LIN {X 0,Y 263.962,Z 436.135,A -85,B 0,C 180,E1 10063.892,E2 10063.892} C_VEL
LIN {X 0,Y 268.762,Z 444.869,A -85,B 0,C 180,E1 10060.552,E2 10060.552} C_VEL
LIN {X 0,Y 273.864,Z 454.801,A -85,B 0,C 180,E1 10057.516,E2 10057.516} C_VEL
LIN {X 0,Y 279.077,Z 465.837,A -85,B 0,C 180,E1 10054.772,E2 10054.772} C_VEL
LIN {X 0,Y 266.38,Z 615.165,A -85,B 0,C 180,E1 10051.274,E2 10051.274} C_VEL
LIN {X 0,Y 262.944,Z 636.67,A -85,B 0,C 180,E1 10050.519,E2 10050.519} C_VEL
LIN {X 0,Y 258.07,Z 657.385,A -85,B 0,C 180,E1 10049.523,E2 10049.523} C_VEL
LIN {X 0,Y 252.139,Z 676.761,A -85,B 0,C 180,E1 10048.274,E2 10048.274} C_VEL
LIN {X 0,Y 244.931,Z 696.333,A -85,B 0,C 180,E1 10046.572,E2 10046.572} C_VEL
LIN {X 0,Y 237.126,Z 714.604,A -85,B 0,C 180,E1 10044.466,E2 10044.466} C_VEL
LIN {X 0,Y 228.803,Z 731.913,A -85,B 0,C 180,E1 10041.866,E2 10041.866} C_VEL
LIN {X 0,Y 220.297,Z 748.012,A -85,B 0,C 180,E1 10038.744,E2 10038.744} C_VEL
LIN {X 0,Y 211.941,Z 762.843,A -85,B 0,C 180,E1 10035.042,E2 10035.042} C_VEL
LIN {X 0,Y 204.052,Z 776.444,A -85,B 0,C 180,E1 10030.668,E2 10030.668} C_VEL
LIN {X 0,Y 197.32,Z 788.149,A -85,B 0,C 180,E1 10025.831,E2 10025.831} C_VEL
LIN {X 0,Y 192.074,Z 797.92,A -85,B 0,C 180,E1 10020.673,E2 10020.673} C_VEL
LIN {X 0,Y 188.152,Z 806.55,A -85,B 0,C 180,E1 10014.822,E2 10014.822} C_VEL
LIN {X 0,Y 185.945,Z 813.61,A -85,B 0,C 180,E1 10008.496,E2 10008.496} C_VEL
LIN {X 0,Y 185.499,Z 818.499,A -85,B 0,C 180,E1 10002.451,E2 10002.451} C_VEL
LIN {X 0,Y 186.162,Z 821.531,A -85,B 0,C 180,E1 9996.786,E2 9996.786} C_VEL
LIN {X 0,Y 186.928,Z 822.719,A -85,B 0,C 180,E1 9992.146,E2 9992.146} C_VEL
LIN {X 0,Y 187.015,Z 822.81,A -85,B 0,C 180,E1 9988.759,E2 9988.759} C_VEL
LIN {X 0,Y 186.446,Z 822.014,A -85,B 0,C 180,E1 9984.769,E2 9984.769} C_VEL
LIN {X 0,Y 185.634,Z 819.662,A -85,B 0,C 180,E1 9979.448,E2 9979.448} C_VEL
LIN {X 0,Y 185.656,Z 815.362,A -85,B 0,C 180,E1 9973.416,E2 9973.416} C_VEL
LIN {X 0,Y 187.283,Z 808.876,A -85,B 0,C 180,E1 9967.063,E2 9967.063} C_VEL
LIN {X 0,Y 190.629,Z 800.812,A -85,B 0,C 180,E1 9961.149,E2 9961.149} C_VEL
LIN {X 0,Y 195.495,Z 791.337,A -85,B 0,C 180,E1 9955.766,E2 9955.766} C_VEL
LIN {X 0,Y 201.572,Z 780.562,A -85,B 0,C 180,E1 9950.954,E2 9950.954} C_VEL
LIN {X 0,Y 209.007,Z 767.743,A -85,B 0,C 180,E1 9946.46,E2 9946.46} C_VEL
LIN {X 0,Y 217.161,Z 753.439,A -85,B 0,C 180,E1 9942.553,E2 9942.553} C_VEL
LIN {X 0,Y 225.436,Z 738.145,A -85,B 0,C 180,E1 9939.292,E2 9939.292} C_VEL
LIN {X 0,Y 233.414,Z 722.238,A -85,B 0,C 180,E1 9936.636,E2 9936.636} C_VEL
LIN {X 0,Y 241.151,Z 705.141,A -85,B 0,C 180,E1 9934.404,E2 9934.404} C_VEL
LIN {X 0,Y 248.509,Z 686.643,A -85,B 0,C 180,E1 9932.554,E2 9932.554} C_VEL
LIN {X 0,Y 255.094,Z 667.118,A -85,B 0,C 180,E1 9931.085,E2 9931.085} C_VEL
LIN {X 0,Y 260.539,Z 647.028,A -85,B 0,C 180,E1 9929.966,E2 9929.966} C_VEL
LIN {X 0,Y 264.728,Z 625.774,A -85,B 0,C 180,E1 9929.09,E2 9929.09} C_VEL
LIN {X 0,Y 267.336,Z 604.079,A -85,B 0,C 180,E1 9928.456,E2 9928.456} C_VEL
LIN {X 0,Y 278.878,Z 465.633,A -85,B 0,C 180,E1 9925.226,E2 9925.226} C_VEL
LIN {X 0,Y 273.338,Z 453.94,A -85,B 0,C 180,E1 9922.303,E2 9922.303} C_VEL
LIN {X 0,Y 267.946,Z 443.512,A -85,B 0,C 180,E1 9919.057,E2 9919.057} C_VEL
LIN {X 0,Y 262.361,Z 433.364,A -85,B 0,C 180,E1 9915.019,E2 9915.019} C_VEL
LIN {X 0,Y 258.426,Z 426.882,A -85,B 0,C 180,E1 9911.493,E2 9911.493} C_VEL
LIN {X 0,Y 256.433,Z 423.717,A -85,B 0,C 180,E1 9909.312,E2 9909.312} C_VEL
LIN {X 0,Y 254.428,Z 420.112,A -85,B 0,C 180,E1 9906.543,E2 9906.543} C_VEL
LIN {X 0,Y 252.019,Z 415.913,A -85,B 0,C 180,E1 9901.364,E2 9901.364} C_VEL
LIN {X 0,Y 251.317,Z 414.93,A -85,B 0,C 180,E1 9895.664,E2 9895.664} C_VEL
LIN {X 0,Y 252.963,Z 416.019,A -85,B 0,C 180,E1 9889.754,E2 9889.754} C_VEL
LIN {X 0,Y 256.776,Z 421.342,A -85,B 0,C 180,E1 9883.95,E2 9883.95} C_VEL
LIN {X 0,Y 260.32,Z 426.562,A -85,B 0,C 180,E1 9880.361,E2 9880.361} C_VEL
LIN {X 0,Y 263.768,Z 431.814,A -85,B 0,C 180,E1 9877.547,E2 9877.547} C_VEL
LIN {X 0,Y 267.986,Z 438.368,A -85,B 0,C 180,E1 9874.65,E2 9874.65} C_VEL
LIN {X 0,Y 273.416,Z 447.764,A -85,B 0,C 180,E1 9871.435,E2 9871.435} C_VEL
LIN {X 0,Y 278.64,Z 457.79,A -85,B 0,C 180,E1 9868.724,E2 9868.724} C_VEL
LIN {X 0,Y 269.524,Z 577.471,A -85,B 0,C 180,E1 9866.054,E2 9866.054} C_VEL
LIN {X 0,Y 267.466,Z 596.812,A -85,B 0,C 180,E1 9865.36,E2 9865.36} C_VEL
LIN {X 0,Y 264.312,Z 615.233,A -85,B 0,C 180,E1 9864.419,E2 9864.419} C_VEL
LIN {X 0,Y 259.903,Z 633.791,A -85,B 0,C 180,E1 9863.145,E2 9863.145} C_VEL
LIN {X 0,Y 254.582,Z 651.308,A -85,B 0,C 180,E1 9861.583,E2 9861.583} C_VEL
LIN {X 0,Y 248.111,Z 668.635,A -85,B 0,C 180,E1 9859.608,E2 9859.608} C_VEL
LIN {X 0,Y 240.971,Z 684.785,A -85,B 0,C 180,E1 9857.257,E2 9857.257} C_VEL
LIN {X 0,Y 233.585,Z 699.288,A -85,B 0,C 180,E1 9854.586,E2 9854.586} C_VEL
LIN {X 0,Y 225.6,Z 713.172,A -85,B 0,C 180,E1 9851.327,E2 9851.327} C_VEL
LIN {X 0,Y 217.777,Z 725.421,A -85,B 0,C 180,E1 9847.634,E2 9847.634} C_VEL
LIN {X 0,Y 210.347,Z 736.116,A -85,B 0,C 180,E1 9843.461,E2 9843.461} C_VEL
LIN {X 0,Y 203.591,Z 745.264,A -85,B 0,C 180,E1 9838.769,E2 9838.769} C_VEL
LIN {X 0,Y 197.74,Z 752.844,A -85,B 0,C 180,E1 9833.544,E2 9833.544} C_VEL
LIN {X 0,Y 193.295,Z 758.557,A -85,B 0,C 180,E1 9828.081,E2 9828.081} C_VEL
LIN {X 0,Y 190.101,Z 762.723,A -85,B 0,C 180,E1 9822.145,E2 9822.145} C_VEL
LIN {X 0,Y 188.303,Z 765.165,A -85,B 0,C 180,E1 9816.096,E2 9816.096} C_VEL
LIN {X 0,Y 187.747,Z 765.976,A -85,B 0,C 180,E1 9810,E2 9810} C_VEL
LIN {X 0,Y 188.29,Z 765.2,A -85,B 0,C 180,E1 9803.904,E2 9803.904} C_VEL
LIN {X 0,Y 190.069,Z 762.799,A -85,B 0,C 180,E1 9797.853,E2 9797.853} C_VEL
LIN {X 0,Y 193.245,Z 758.673,A -85,B 0,C 180,E1 9791.915,E2 9791.915} C_VEL
LIN {X 0,Y 197.948,Z 752.674,A -85,B 0,C 180,E1 9786.167,E2 9786.167} C_VEL
LIN {X 0,Y 203.857,Z 745.036,A -85,B 0,C 180,E1 9780.951,E2 9780.951} C_VEL
LIN {X 0,Y 210.664,Z 735.828,A -85,B 0,C 180,E1 9776.269,E2 9776.269} C_VEL
LIN {X 0,Y 218.141,Z 725.064,A -85,B 0,C 180,E1 9772.108,E2 9772.108} C_VEL
LIN {X 0,Y 226.001,Z 712.736,A -85,B 0,C 180,E1 9768.425,E2 9768.425} C_VEL
LIN {X 0,Y 234.026,Z 698.729,A -85,B 0,C 180,E1 9765.172,E2 9765.172} C_VEL
LIN {X 0,Y 241.439,Z 684.148,A -85,B 0,C 180,E1 9762.513,E2 9762.513} C_VEL
LIN {X 0,Y 248.603,Z 667.849,A -85,B 0,C 180,E1 9760.17,E2 9760.17} C_VEL
LIN {X 0,Y 255.089,Z 650.314,A -85,B 0,C 180,E1 9758.199,E2 9758.199} C_VEL
LIN {X 0,Y 260.429,Z 632.572,A -85,B 0,C 180,E1 9756.641,E2 9756.641} C_VEL
LIN {X 0,Y 264.883,Z 613.37,A -85,B 0,C 180,E1 9755.356,E2 9755.356} C_VEL
LIN {X 0,Y 268.08,Z 593.774,A -85,B 0,C 180,E1 9754.394,E2 9754.394} C_VEL
LIN {X 0,Y 270.011,Z 573.44,A -85,B 0,C 180,E1 9753.717,E2 9753.717} C_VEL
LIN {X 0,Y 278.808,Z 457.69,A -85,B 0,C 180,E1 9751.152,E2 9751.152} C_VEL
LIN {X 0,Y 272.497,Z 445.95,A -85,B 0,C 180,E1 9747.839,E2 9747.839} C_VEL
LIN {X 0,Y 267.272,Z 437.11,A -85,B 0,C 180,E1 9744.653,E2 9744.653} C_VEL
LIN {X 0,Y 262.532,Z 429.641,A -85,B 0,C 180,E1 9741.212,E2 9741.212} C_VEL
LIN {X 0,Y 259.127,Z 424.746,A -85,B 0,C 180,E1 9738.213,E2 9738.213} C_VEL
LIN {X 0,Y 256.354,Z 420.667,A -85,B 0,C 180,E1 9735.149,E2 9735.149} C_VEL
LIN {X 0,Y 253.062,Z 416.095,A -85,B 0,C 180,E1 9729.782,E2 9729.782} C_VEL
LIN {X 0,Y 251.573,Z 415.164,A -85,B 0,C 180,E1 9723.875,E2 9723.875} C_VEL
LIN {X 0,Y 252.355,Z 416.185,A -85,B 0,C 180,E1 9718.411,E2 9718.411} C_VEL
LIN {X 0,Y 255.115,Z 421.076,A -85,B 0,C 180,E1 9712.796,E2 9712.796} C_VEL
LIN {X 0,Y 258.442,Z 426.742,A -85,B 0,C 180,E1 9708.734,E2 9708.734} C_VEL
LIN {X 0,Y 261.024,Z 431.187,A -85,B 0,C 180,E1 9706.272,E2 9706.272} C_VEL
LIN {X 0,Y 262.586,Z 435.115,A -85,B 0,C 180,E1 9704.85,E2 9704.85} C_VEL
LIN {X 0,Y 264.574,Z 443.488,A -85,B 0,C 180,E1 9702.933,E2 9702.933} C_VEL
LIN {X 0,Y 266.814,Z 452.064,A -85,B 0,C 180,E1 9701.05,E2 9701.05} C_VEL
LIN {X 0,Y 267.623,Z 454.063,A -85,B 0,C 180,E1 9700.49,E2 9700.49} C_VEL
LIN {X 0,Y 272.716,Z 464.616,A -85,B 0,C 180,E1 9697.416,E2 9697.416} C_VEL
LIN {X 0,Y 274.98,Z 470.078,A -85,B 0,C 180,E1 9696.14,E2 9696.14} C_VEL
LIN {X 0,Y 262.311,Z 614.422,A -85,B 0,C 180,E1 9692.779,E2 9692.779} C_VEL
LIN {X 0,Y 258.795,Z 635.834,A -85,B 0,C 180,E1 9692.035,E2 9692.035} C_VEL
LIN {X 0,Y 253.894,Z 656.209,A -85,B 0,C 180,E1 9691.07,E2 9691.07} C_VEL
LIN {X 0,Y 247.581,Z 676.274,A -85,B 0,C 180,E1 9689.793,E2 9689.793} C_VEL
LIN {X 0,Y 240.198,Z 695.651,A -85,B 0,C 180,E1 9688.12,E2 9688.12} C_VEL
LIN {X 0,Y 232.104,Z 713.934,A -85,B 0,C 180,E1 9686.019,E2 9686.019} C_VEL
LIN {X 0,Y 223.481,Z 731.176,A -85,B 0,C 180,E1 9683.423,E2 9683.423} C_VEL
LIN {X 0,Y 214.547,Z 747.362,A -85,B 0,C 180,E1 9680.258,E2 9680.258} C_VEL
LIN {X 0,Y 205.621,Z 762.427,A -85,B 0,C 180,E1 9676.428,E2 9676.428} C_VEL
LIN {X 0,Y 197.354,Z 775.9,A -85,B 0,C 180,E1 9671.969,E2 9671.969} C_VEL
LIN {X 0,Y 190.055,Z 787.822,A -85,B 0,C 180,E1 9666.85,E2 9666.85} C_VEL
LIN {X 0,Y 184.137,Z 798.176,A -85,B 0,C 180,E1 9661.053,E2 9661.053} C_VEL
LIN {X 0,Y 180.13,Z 806.495,A -85,B 0,C 180,E1 9654.951,E2 9654.951} C_VEL
LIN {X 0,Y 177.989,Z 812.955,A -85,B 0,C 180,E1 9648.674,E2 9648.674} C_VEL
LIN {X 0,Y 177.55,Z 817.657,A -85,B 0,C 180,E1 9642.356,E2 9642.356} C_VEL
LIN {X 0,Y 178.282,Z 820.523,A -85,B 0,C 180,E1 9636.44,E2 9636.44} C_VEL
LIN {X 0,Y 179.036,Z 821.548,A -85,B 0,C 180,E1 9631.92,E2 9631.92} C_VEL
LIN {X 0,Y 179.07,Z 821.577,A -85,B 0,C 180,E1 9628.4,E2 9628.4} C_VEL
LIN {X 0,Y 178.404,Z 820.702,A -85,B 0,C 180,E1 9624.21,E2 9624.21} C_VEL
LIN {X 0,Y 177.589,Z 818.027,A -85,B 0,C 180,E1 9618.306,E2 9618.306} C_VEL
LIN {X 0,Y 177.869,Z 813.516,A -85,B 0,C 180,E1 9611.991,E2 9611.991} C_VEL
LIN {X 0,Y 179.816,Z 807.245,A -85,B 0,C 180,E1 9605.703,E2 9605.703} C_VEL
LIN {X 0,Y 183.877,Z 798.609,A -85,B 0,C 180,E1 9599.261,E2 9599.261} C_VEL
LIN {X 0,Y 189.692,Z 788.341,A -85,B 0,C 180,E1 9593.445,E2 9593.445} C_VEL
LIN {X 0,Y 196.965,Z 776.407,A -85,B 0,C 180,E1 9588.263,E2 9588.263} C_VEL
LIN {X 0,Y 205.148,Z 763.047,A -85,B 0,C 180,E1 9583.795,E2 9583.795} C_VEL
LIN {X 0,Y 213.949,Z 748.192,A -85,B 0,C 180,E1 9579.968,E2 9579.968} C_VEL
LIN {X 0,Y 222.83,Z 732.143,A -85,B 0,C 180,E1 9576.782,E2 9576.782} C_VEL
LIN {X 0,Y 231.368,Z 715.151,A -85,B 0,C 180,E1 9574.18,E2 9574.18} C_VEL
LIN {X 0,Y 239.105,Z 697.83,A -85,B 0,C 180,E1 9572.138,E2 9572.138} C_VEL
LIN {X 0,Y 246.063,Z 679.96,A -85,B 0,C 180,E1 9570.524,E2 9570.524} C_VEL
LIN {X 0,Y 252.141,Z 661.532,A -85,B 0,C 180,E1 9569.264,E2 9569.264} C_VEL
LIN {X 0,Y 257.488,Z 640.986,A -85,B 0,C 180,E1 9568.212,E2 9568.212} C_VEL
LIN {X 0,Y 261.349,Z 619.931,A -85,B 0,C 180,E1 9567.418,E2 9567.418} C_VEL
LIN {X 0,Y 264.036,Z 594.652,A -85,B 0,C 180,E1 9566.746,E2 9566.746} C_VEL
LIN {X 0,Y 274.757,Z 469.441,A -85,B 0,C 180,E1 9563.824,E2 9563.824} C_VEL
LIN {X 0,Y 269.41,Z 457.799,A -85,B 0,C 180,E1 9560.758,E2 9560.758} C_VEL
LIN {X 0,Y 263.947,Z 447.113,A -85,B 0,C 180,E1 9557.129,E2 9557.129} C_VEL
LIN {X 0,Y 259.778,Z 439.543,A -85,B 0,C 180,E1 9553.805,E2 9553.805} C_VEL
LIN {X 0,Y 256.77,Z 434.226,A -85,B 0,C 180,E1 9550.886,E2 9550.886} C_VEL
LIN {X 0,Y 253.434,Z 428.163,A -85,B 0,C 180,E1 9546.569,E2 9546.569} C_VEL
LIN {X 0,Y 250.96,Z 423.8,A -85,B 0,C 180,E1 9541.141,E2 9541.141} C_VEL
LIN {X 0,Y 250.345,Z 422.871,A -85,B 0,C 180,E1 9535.647,E2 9535.647} C_VEL
LIN {X 0,Y 252.001,Z 423.991,A -85,B 0,C 180,E1 9529.714,E2 9529.714} C_VEL
LIN {X 0,Y 255.526,Z 429.237,A -85,B 0,C 180,E1 9524.219,E2 9524.219} C_VEL
LIN {X 0,Y 258.761,Z 434.142,A -85,B 0,C 180,E1 9520.825,E2 9520.825} C_VEL
LIN {X 0,Y 262.133,Z 439.449,A -85,B 0,C 180,E1 9517.971,E2 9517.971} C_VEL
LIN {X 0,Y 266.367,Z 446.383,A -85,B 0,C 180,E1 9514.961,E2 9514.961} C_VEL
LIN {X 0,Y 271.172,Z 455.032,A -85,B 0,C 180,E1 9512.017,E2 9512.017} C_VEL
LIN {X 0,Y 274.626,Z 461.918,A -85,B 0,C 180,E1 9510.11,E2 9510.11} C_VEL
LIN {X 0,Y 265.44,Z 578.24,A -85,B 0,C 180,E1 9507.518,E2 9507.518} C_VEL
LIN {X 0,Y 263.304,Z 597.581,A -85,B 0,C 180,E1 9506.825,E2 9506.825} C_VEL
LIN {X 0,Y 260.034,Z 616.06,A -85,B 0,C 180,E1 9505.886,E2 9505.886} C_VEL
LIN {X 0,Y 255.561,Z 634.361,A -85,B 0,C 180,E1 9504.639,E2 9504.639} C_VEL
LIN {X 0,Y 250.09,Z 651.862,A -85,B 0,C 180,E1 9503.09,E2 9503.09} C_VEL
LIN {X 0,Y 243.394,Z 669.282,A -85,B 0,C 180,E1 9501.118,E2 9501.118} C_VEL
LIN {X 0,Y 235.981,Z 685.526,A -85,B 0,C 180,E1 9498.762,E2 9498.762} C_VEL
LIN {X 0,Y 228.025,Z 700.565,A -85,B 0,C 180,E1 9495.98,E2 9495.98} C_VEL
LIN {X 0,Y 219.721,Z 714.42,A -85,B 0,C 180,E1 9492.689,E2 9492.689} C_VEL
LIN {X 0,Y 211.561,Z 726.652,A -85,B 0,C 180,E1 9488.944,E2 9488.944} C_VEL
LIN {X 0,Y 203.781,Z 737.336,A -85,B 0,C 180,E1 9484.69,E2 9484.69} C_VEL
LIN {X 0,Y 196.675,Z 746.477,A -85,B 0,C 180,E1 9479.881,E2 9479.881} C_VEL
LIN {X 0,Y 190.493,Z 754.053,A -85,B 0,C 180,E1 9474.497,E2 9474.497} C_VEL
LIN {X 0,Y 185.77,Z 759.763,A -85,B 0,C 180,E1 9468.84,E2 9468.84} C_VEL
LIN {X 0,Y 182.363,Z 763.927,A -85,B 0,C 180,E1 9462.668,E2 9462.668} C_VEL
LIN {X 0,Y 180.435,Z 766.367,A -85,B 0,C 180,E1 9456.363,E2 9456.363} C_VEL
LIN {X 0,Y 179.838,Z 767.178,A -85,B 0,C 180,E1 9450,E2 9450} C_VEL
LIN {X 0,Y 180.422,Z 766.402,A -85,B 0,C 180,E1 9443.637,E2 9443.637} C_VEL
LIN {X 0,Y 182.33,Z 764.002,A -85,B 0,C 180,E1 9437.329,E2 9437.329} C_VEL
LIN {X 0,Y 185.719,Z 759.877,A -85,B 0,C 180,E1 9431.155,E2 9431.155} C_VEL
LIN {X 0,Y 190.717,Z 753.881,A -85,B 0,C 180,E1 9425.203,E2 9425.203} C_VEL
LIN {X 0,Y 196.958,Z 746.25,A -85,B 0,C 180,E1 9419.831,E2 9419.831} C_VEL
LIN {X 0,Y 204.119,Z 737.048,A -85,B 0,C 180,E1 9415.034,E2 9415.034} C_VEL
LIN {X 0,Y 211.947,Z 726.296,A -85,B 0,C 180,E1 9410.793,E2 9410.793} C_VEL
LIN {X 0,Y 220.146,Z 713.986,A -85,B 0,C 180,E1 9407.059,E2 9407.059} C_VEL
LIN {X 0,Y 228.485,Z 700.025,A -85,B 0,C 180,E1 9403.778,E2 9403.778} C_VEL
LIN {X 0,Y 236.481,Z 684.837,A -85,B 0,C 180,E1 9401.002,E2 9401.002} C_VEL
LIN {X 0,Y 243.906,Z 668.454,A -85,B 0,C 180,E1 9398.657,E2 9398.657} C_VEL
LIN {X 0,Y 250.266,Z 651.876,A -85,B 0,C 180,E1 9396.793,E2 9396.793} C_VEL
LIN {X 0,Y 255.814,Z 634.148,A -85,B 0,C 180,E1 9395.228,E2 9395.228} C_VEL
LIN {X 0,Y 260.374,Z 615.388,A -85,B 0,C 180,E1 9393.96,E2 9393.96} C_VEL
LIN {X 0,Y 263.777,Z 595.743,A -85,B 0,C 180,E1 9392.979,E2 9392.979} C_VEL
LIN {X 0,Y 265.852,Z 575.618,A -85,B 0,C 180,E1 9392.291,E2 9392.291} C_VEL
LIN {X 0,Y 274.724,Z 461.747,A -85,B 0,C 180,E1 9389.729,E2 9389.729} C_VEL
LIN {X 0,Y 269.186,Z 451.135,A -85,B 0,C 180,E1 9386.589,E2 9386.589} C_VEL
LIN {X 0,Y 264.409,Z 442.959,A -85,B 0,C 180,E1 9383.454,E2 9383.454} C_VEL
LIN {X 0,Y 260.148,Z 436.17,A -85,B 0,C 180,E1 9380.12,E2 9380.12} C_VEL
LIN {X 0,Y 257.621,Z 432.313,A -85,B 0,C 180,E1 9377.739,E2 9377.739} C_VEL
LIN {X 0,Y 255.045,Z 428.396,A -85,B 0,C 180,E1 9374.763,E2 9374.763} C_VEL
LIN {X 0,Y 252.008,Z 423.989,A -85,B 0,C 180,E1 9369.593,E2 9369.593} C_VEL
LIN {X 0,Y 250.592,Z 423.106,A -85,B 0,C 180,E1 9363.661,E2 9363.661} C_VEL
LIN {X 0,Y 251.362,Z 424.279,A -85,B 0,C 180,E1 9358.405,E2 9358.405} C_VEL
LIN {X 0,Y 253.873,Z 428.918,A -85,B 0,C 180,E1 9353.101,E2 9353.101} C_VEL
LIN {X 0,Y 256.901,Z 434.265,A -85,B 0,C 180,E1 9349.233,E2 9349.233} C_VEL
LIN {X 0,Y 260.684,Z 440.814,A -85,B 0,C 180,E1 9345.621,E2 9345.621} C_VEL
LIN {X 0,Y 265.967,Z 450.804,A -85,B 0,C 180,E1 9341.592,E2 9341.592} C_VEL
LIN {X 0,Y 267.623,Z 454.063,A -85,B 0,C 180,E1 9340.49,E2 9340.49} C_VEL
LIN {X 0,Y 268.653,Z 457.702,A -85,B 0,C 180,E1 9339.728,E2 9339.728} C_VEL
LIN {X 0,Y 270.267,Z 470.787,A -85,B 0,C 180,E1 9338.119,E2 9338.119} C_VEL
LIN {X 0,Y 271.051,Z 473.538,A -85,B 0,C 180,E1 9337.597,E2 9337.597} C_VEL
LIN {X 0,Y 258.457,Z 613.492,A -85,B 0,C 180,E1 9334.336,E2 9334.336} C_VEL
LIN {X 0,Y 254.871,Z 634.831,A -85,B 0,C 180,E1 9333.607,E2 9333.607} C_VEL
LIN {X 0,Y 249.872,Z 655.168,A -85,B 0,C 180,E1 9332.661,E2 9332.661} C_VEL
LIN {X 0,Y 243.592,Z 674.701,A -85,B 0,C 180,E1 9331.446,E2 9331.446} C_VEL
LIN {X 0,Y 235.986,Z 694.185,A -85,B 0,C 180,E1 9329.804,E2 9329.804} C_VEL
LIN {X 0,Y 227.614,Z 712.526,A -85,B 0,C 180,E1 9327.735,E2 9327.735} C_VEL
LIN {X 0,Y 218.527,Z 730.074,A -85,B 0,C 180,E1 9325.116,E2 9325.116} C_VEL
LIN {X 0,Y 209.154,Z 746.368,A -85,B 0,C 180,E1 9321.926,E2 9321.926} C_VEL
LIN {X 0,Y 199.978,Z 761.113,A -85,B 0,C 180,E1 9318.155,E2 9318.155} C_VEL
LIN {X 0,Y 191.242,Z 774.603,A -85,B 0,C 180,E1 9313.639,E2 9313.639} C_VEL
LIN {X 0,Y 183.44,Z 786.534,A -85,B 0,C 180,E1 9308.415,E2 9308.415} C_VEL
LIN {X 0,Y 177.041,Z 796.897,A -85,B 0,C 180,E1 9302.446,E2 9302.446} C_VEL
LIN {X 0,Y 172.62,Z 805.225,A -85,B 0,C 180,E1 9296.116,E2 9296.116} C_VEL
LIN {X 0,Y 170.181,Z 811.698,A -85,B 0,C 180,E1 9289.565,E2 9289.565} C_VEL
LIN {X 0,Y 169.577,Z 816.415,A -85,B 0,C 180,E1 9282.947,E2 9282.947} C_VEL
LIN {X 0,Y 170.287,Z 819.301,A -85,B 0,C 180,E1 9276.744,E2 9276.744} C_VEL
LIN {X 0,Y 171.107,Z 820.343,A -85,B 0,C 180,E1 9272.009,E2 9272.009} C_VEL
LIN {X 0,Y 171.178,Z 820.405,A -85,B 0,C 180,E1 9268.661,E2 9268.661} C_VEL
LIN {X 0,Y 170.476,Z 819.577,A -85,B 0,C 180,E1 9264.278,E2 9264.278} C_VEL
LIN {X 0,Y 169.621,Z 816.985,A -85,B 0,C 180,E1 9258.094,E2 9258.094} C_VEL
LIN {X 0,Y 169.97,Z 812.559,A -85,B 0,C 180,E1 9251.479,E2 9251.479} C_VEL
LIN {X 0,Y 172.273,Z 805.975,A -85,B 0,C 180,E1 9244.566,E2 9244.566} C_VEL
LIN {X 0,Y 176.757,Z 797.329,A -85,B 0,C 180,E1 9237.879,E2 9237.879} C_VEL
LIN {X 0,Y 183.113,Z 786.955,A -85,B 0,C 180,E1 9231.839,E2 9231.839} C_VEL
LIN {X 0,Y 190.759,Z 775.213,A -85,B 0,C 180,E1 9226.637,E2 9226.637} C_VEL
LIN {X 0,Y 199.421,Z 761.827,A -85,B 0,C 180,E1 9222.096,E2 9222.096} C_VEL
LIN {X 0,Y 208.727,Z 746.868,A -85,B 0,C 180,E1 9218.225,E2 9218.225} C_VEL
LIN {X 0,Y 217.99,Z 730.79,A -85,B 0,C 180,E1 9215.045,E2 9215.045} C_VEL
LIN {X 0,Y 226.895,Z 713.67,A -85,B 0,C 180,E1 9212.45,E2 9212.45} C_VEL
LIN {X 0,Y 235.227,Z 695.538,A -85,B 0,C 180,E1 9210.362,E2 9210.362} C_VEL
LIN {X 0,Y 242.416,Z 677.385,A -85,B 0,C 180,E1 9208.784,E2 9208.784} C_VEL
LIN {X 0,Y 248.711,Z 658.403,A -85,B 0,C 180,E1 9207.548,E2 9207.548} C_VEL
LIN {X 0,Y 253.921,Z 638.253,A -85,B 0,C 180,E1 9206.563,E2 9206.563} C_VEL
LIN {X 0,Y 257.673,Z 617.588,A -85,B 0,C 180,E1 9205.814,E2 9205.814} C_VEL
LIN {X 0,Y 260.622,Z 589.211,A -85,B 0,C 180,E1 9205.086,E2 9205.086} C_VEL
LIN {X 0,Y 270.847,Z 473.338,A -85,B 0,C 180,E1 9202.405,E2 9202.405} C_VEL
LIN {X 0,Y 266.038,Z 462.77,A -85,B 0,C 180,E1 9199.427,E2 9199.427} C_VEL
LIN {X 0,Y 261.467,Z 453.484,A -85,B 0,C 180,E1 9196.152,E2 9196.152} C_VEL
LIN {X 0,Y 257.896,Z 446.68,A -85,B 0,C 180,E1 9193.109,E2 9193.109} C_VEL
LIN {X 0,Y 254.958,Z 441.205,A -85,B 0,C 180,E1 9190.05,E2 9190.05} C_VEL
LIN {X 0,Y 251.865,Z 435.512,A -85,B 0,C 180,E1 9185.695,E2 9185.695} C_VEL
LIN {X 0,Y 249.905,Z 431.687,A -85,B 0,C 180,E1 9180.917,E2 9180.917} C_VEL
LIN {X 0,Y 249.389,Z 430.818,A -85,B 0,C 180,E1 9175.4,E2 9175.4} C_VEL
LIN {X 0,Y 250.937,Z 431.891,A -85,B 0,C 180,E1 9169.902,E2 9169.902} C_VEL
LIN {X 0,Y 254.192,Z 436.961,A -85,B 0,C 180,E1 9164.602,E2 9164.602} C_VEL
LIN {X 0,Y 257.218,Z 441.719,A -85,B 0,C 180,E1 9161.295,E2 9161.295} C_VEL
LIN {X 0,Y 260.737,Z 447.429,A -85,B 0,C 180,E1 9158.221,E2 9158.221} C_VEL
LIN {X 0,Y 265.223,Z 455.175,A -85,B 0,C 180,E1 9154.965,E2 9154.965} C_VEL
LIN {X 0,Y 270.149,Z 464.689,A -85,B 0,C 180,E1 9151.902,E2 9151.902} C_VEL
LIN {X 0,Y 270.764,Z 466.184,A -85,B 0,C 180,E1 9151.534,E2 9151.534} C_VEL
LIN {X 0,Y 261.543,Z 578.893,A -85,B 0,C 180,E1 9149.031,E2 9149.031} C_VEL
LIN {X 0,Y 259.335,Z 598.253,A -85,B 0,C 180,E1 9148.341,E2 9148.341} C_VEL
LIN {X 0,Y 256.033,Z 616.456,A -85,B 0,C 180,E1 9147.426,E2 9147.426} C_VEL
LIN {X 0,Y 251.465,Z 634.7,A -85,B 0,C 180,E1 9146.2,E2 9146.2} C_VEL
LIN {X 0,Y 245.442,Z 653.314,A -85,B 0,C 180,E1 9144.559,E2 9144.559} C_VEL
LIN {X 0,Y 238.524,Z 670.647,A -85,B 0,C 180,E1 9142.592,E2 9142.592} C_VEL
LIN {X 0,Y 230.865,Z 686.815,A -85,B 0,C 180,E1 9140.239,E2 9140.239} C_VEL
LIN {X 0,Y 222.606,Z 701.837,A -85,B 0,C 180,E1 9137.443,E2 9137.443} C_VEL
LIN {X 0,Y 213.973,Z 715.667,A -85,B 0,C 180,E1 9134.125,E2 9134.125} C_VEL
LIN {X 0,Y 205.461,Z 727.883,A -85,B 0,C 180,E1 9130.332,E2 9130.332} C_VEL
LIN {X 0,Y 197.315,Z 738.556,A -85,B 0,C 180,E1 9126.001,E2 9126.001} C_VEL
LIN {X 0,Y 189.838,Z 747.69,A -85,B 0,C 180,E1 9121.074,E2 9121.074} C_VEL
LIN {X 0,Y 183.302,Z 755.261,A -85,B 0,C 180,E1 9115.525,E2 9115.525} C_VEL
LIN {X 0,Y 178.101,Z 761.156,A -85,B 0,C 180,E1 9109.41,E2 9109.41} C_VEL
LIN {X 0,Y 174.64,Z 765.131,A -85,B 0,C 180,E1 9103.239,E2 9103.239} C_VEL
LIN {X 0,Y 172.572,Z 767.569,A -85,B 0,C 180,E1 9096.654,E2 9096.654} C_VEL
LIN {X 0,Y 171.929,Z 768.379,A -85,B 0,C 180,E1 9090,E2 9090} C_VEL
LIN {X 0,Y 172.558,Z 767.603,A -85,B 0,C 180,E1 9083.345,E2 9083.345} C_VEL
LIN {X 0,Y 174.606,Z 765.204,A -85,B 0,C 180,E1 9076.759,E2 9076.759} C_VEL
LIN {X 0,Y 178.23,Z 761.081,A -85,B 0,C 180,E1 9070.331,E2 9070.331} C_VEL
LIN {X 0,Y 183.543,Z 755.089,A -85,B 0,C 180,E1 9064.165,E2 9064.165} C_VEL
LIN {X 0,Y 190.141,Z 747.462,A -85,B 0,C 180,E1 9058.629,E2 9058.629} C_VEL
LIN {X 0,Y 197.674,Z 738.268,A -85,B 0,C 180,E1 9053.716,E2 9053.716} C_VEL
LIN {X 0,Y 205.871,Z 727.526,A -85,B 0,C 180,E1 9049.4,E2 9049.4} C_VEL
LIN {X 0,Y 214.422,Z 715.233,A -85,B 0,C 180,E1 9045.618,E2 9045.618} C_VEL
LIN {X 0,Y 223.091,Z 701.302,A -85,B 0,C 180,E1 9042.313,E2 9042.313} C_VEL
LIN {X 0,Y 231.381,Z 686.158,A -85,B 0,C 180,E1 9039.527,E2 9039.527} C_VEL
LIN {X 0,Y 239.064,Z 669.839,A -85,B 0,C 180,E1 9037.182,E2 9037.182} C_VEL
LIN {X 0,Y 245.998,Z 652.299,A -85,B 0,C 180,E1 9035.22,E2 9035.22} C_VEL
LIN {X 0,Y 251.698,Z 634.574,A -85,B 0,C 180,E1 9033.674,E2 9033.674} C_VEL
LIN {X 0,Y 256.472,Z 615.362,A -85,B 0,C 180,E1 9032.396,E2 9032.396} C_VEL
LIN {X 0,Y 259.942,Z 595.562,A -85,B 0,C 180,E1 9031.429,E2 9031.429} C_VEL
LIN {X 0,Y 262.042,Z 575.244,A -85,B 0,C 180,E1 9030.751,E2 9030.751} C_VEL
LIN {X 0,Y 270.904,Z 465.97,A -85,B 0,C 180,E1 9028.313,E2 9028.313} C_VEL
LIN {X 0,Y 265.845,Z 456.132,A -85,B 0,C 180,E1 9025.211,E2 9025.211} C_VEL
LIN {X 0,Y 261.321,Z 448.177,A -85,B 0,C 180,E1 9021.964,E2 9021.964} C_VEL
LIN {X 0,Y 257.639,Z 442.271,A -85,B 0,C 180,E1 9018.791,E2 9018.791} C_VEL
LIN {X 0,Y 255.622,Z 439.169,A -85,B 0,C 180,E1 9016.708,E2 9016.708} C_VEL
LIN {X 0,Y 253.747,Z 436.123,A -85,B 0,C 180,E1 9014.374,E2 9014.374} C_VEL
LIN {X 0,Y 250.952,Z 431.883,A -85,B 0,C 180,E1 9009.402,E2 9009.402} C_VEL
LIN {X 0,Y 249.613,Z 431.063,A -85,B 0,C 180,E1 9003.445,E2 9003.445} C_VEL
LIN {X 0,Y 250.31,Z 432.173,A -85,B 0,C 180,E1 8998.627,E2 8998.627} C_VEL
LIN {X 0,Y 252.595,Z 436.657,A -85,B 0,C 180,E1 8993.482,E2 8993.482} C_VEL
LIN {X 0,Y 255.473,Z 441.965,A -85,B 0,C 180,E1 8989.629,E2 8989.629} C_VEL
LIN {X 0,Y 259.181,Z 448.801,A -85,B 0,C 180,E1 8985.934,E2 8985.934} C_VEL
LIN {X 0,Y 263.838,Z 457.95,A -85,B 0,C 180,E1 8982.238,E2 8982.238} C_VEL
LIN {X 0,Y 268.608,Z 468.029,A -85,B 0,C 180,E1 8979.063,E2 8979.063} C_VEL
LIN {X 0,Y 271.051,Z 473.538,A -85,B 0,C 180,E1 8977.597,E2 8977.597} C_VEL
LIN {X 0,Y 271.539,Z 476.413,A -85,B 0,C 180,E1 8977.208,E2 8977.208} C_VEL
LIN {X 0,Y 271.269,Z 480.92,A -85,B 0,C 180,E1 8977.051,E2 8977.051} C_VEL
LIN {X 0,Y 269.93,Z 487.325,A -85,B 0,C 180,E1 8977.239,E2 8977.239} C_VEL
LIN {X 0,Y 265.57,Z 502.194,A -85,B 0,C 180,E1 8978.257,E2 8978.257} C_VEL
LIN {X 0,Y 264.534,Z 508.324,A -85,B 0,C 180,E1 8978.34,E2 8978.34} C_VEL
LIN {X 0,Y 254.757,Z 612.84,A -85,B 0,C 180,E1 8975.931,E2 8975.931} C_VEL
LIN {X 0,Y 251.088,Z 634.078,A -85,B 0,C 180,E1 8975.216,E2 8975.216} C_VEL
LIN {X 0,Y 245.844,Z 654.788,A -85,B 0,C 180,E1 8974.266,E2 8974.266} C_VEL
LIN {X 0,Y 239.415,Z 674.224,A -85,B 0,C 180,E1 8973.075,E2 8973.075} C_VEL
LIN {X 0,Y 231.603,Z 693.598,A -85,B 0,C 180,E1 8971.463,E2 8971.463} C_VEL
LIN {X 0,Y 222.975,Z 711.859,A -85,B 0,C 180,E1 8969.422,E2 8969.422} C_VEL
LIN {X 0,Y 213.717,Z 729.073,A -85,B 0,C 180,E1 8966.868,E2 8966.868} C_VEL
LIN {X 0,Y 204.038,Z 745.225,A -85,B 0,C 180,E1 8963.715,E2 8963.715} C_VEL
LIN {X 0,Y 194.533,Z 759.801,A -85,B 0,C 180,E1 8959.979,E2 8959.979} C_VEL
LIN {X 0,Y 185.3,Z 773.305,A -85,B 0,C 180,E1 8955.417,E2 8955.417} C_VEL
LIN {X 0,Y 176.976,Z 785.247,A -85,B 0,C 180,E1 8950.094,E2 8950.094} C_VEL
LIN {X 0,Y 170.06,Z 795.62,A -85,B 0,C 180,E1 8943.954,E2 8943.954} C_VEL
LIN {X 0,Y 165.185,Z 803.954,A -85,B 0,C 180,E1 8937.388,E2 8937.388} C_VEL
LIN {X 0,Y 162.407,Z 810.439,A -85,B 0,C 180,E1 8930.543,E2 8930.543} C_VEL
LIN {X 0,Y 161.613,Z 815.173,A -85,B 0,C 180,E1 8923.597,E2 8923.597} C_VEL
LIN {X 0,Y 162.282,Z 818.076,A -85,B 0,C 180,E1 8917.078,E2 8917.078} C_VEL
LIN {X 0,Y 163.175,Z 819.137,A -85,B 0,C 180,E1 8912.107,E2 8912.107} C_VEL
LIN {X 0,Y 163.256,Z 819.202,A -85,B 0,C 180,E1 8908.596,E2 8908.596} C_VEL
LIN {X 0,Y 162.481,Z 818.356,A -85,B 0,C 180,E1 8903.995,E2 8903.995} C_VEL
LIN {X 0,Y 161.638,Z 815.742,A -85,B 0,C 180,E1 8897.497,E2 8897.497} C_VEL
LIN {X 0,Y 162.159,Z 811.3,A -85,B 0,C 180,E1 8890.552,E2 8890.552} C_VEL
LIN {X 0,Y 164.796,Z 804.703,A -85,B 0,C 180,E1 8883.323,E2 8883.323} C_VEL
LIN {X 0,Y 169.748,Z 796.048,A -85,B 0,C 180,E1 8876.381,E2 8876.381} C_VEL
LIN {X 0,Y 176.556,Z 785.763,A -85,B 0,C 180,E1 8870.215,E2 8870.215} C_VEL
LIN {X 0,Y 184.79,Z 773.917,A -85,B 0,C 180,E1 8864.863,E2 8864.863} C_VEL
LIN {X 0,Y 193.946,Z 760.519,A -85,B 0,C 180,E1 8860.273,E2 8860.273} C_VEL
LIN {X 0,Y 203.708,Z 745.539,A -85,B 0,C 180,E1 8856.396,E2 8856.396} C_VEL
LIN {X 0,Y 213.209,Z 729.692,A -85,B 0,C 180,E1 8853.276,E2 8853.276} C_VEL
LIN {X 0,Y 222.597,Z 712.279,A -85,B 0,C 180,E1 8850.666,E2 8850.666} C_VEL
LIN {X 0,Y 231.206,Z 694.085,A -85,B 0,C 180,E1 8848.615,E2 8848.615} C_VEL
LIN {X 0,Y 238.607,Z 675.837,A -85,B 0,C 180,E1 8847.072,E2 8847.072} C_VEL
LIN {X 0,Y 245.023,Z 656.831,A -85,B 0,C 180,E1 8845.873,E2 8845.873} C_VEL
LIN {X 0,Y 250.242,Z 636.931,A -85,B 0,C 180,E1 8844.927,E2 8844.927} C_VEL
LIN {X 0,Y 254.035,Z 616.367,A -85,B 0,C 180,E1 8844.2,E2 8844.2} C_VEL
LIN {X 0,Y 257.092,Z 587.514,A -85,B 0,C 180,E1 8843.472,E2 8843.472} C_VEL
LIN {X 0,Y 267.095,Z 477.349,A -85,B 0,C 180,E1 8840.946,E2 8840.946} C_VEL
LIN {X 0,Y 262.464,Z 466.849,A -85,B 0,C 180,E1 8837.801,E2 8837.801} C_VEL
LIN {X 0,Y 257.967,Z 457.509,A -85,B 0,C 180,E1 8834.19,E2 8834.19} C_VEL
LIN {X 0,Y 254.309,Z 450.317,A -85,B 0,C 180,E1 8830.534,E2 8830.534} C_VEL
LIN {X 0,Y 252.182,Z 446.451,A -85,B 0,C 180,E1 8827.861,E2 8827.861} C_VEL
LIN {X 0,Y 250.603,Z 443.213,A -85,B 0,C 180,E1 8825.265,E2 8825.265} C_VEL
LIN {X 0,Y 248.856,Z 439.575,A -85,B 0,C 180,E1 8820.69,E2 8820.69} C_VEL
LIN {X 0,Y 248.41,Z 438.758,A -85,B 0,C 180,E1 8815.382,E2 8815.382} C_VEL
LIN {X 0,Y 249.865,Z 439.829,A -85,B 0,C 180,E1 8810.091,E2 8810.091} C_VEL
LIN {X 0,Y 252.865,Z 444.683,A -85,B 0,C 180,E1 8804.989,E2 8804.989} C_VEL
LIN {X 0,Y 255.69,Z 449.295,A -85,B 0,C 180,E1 8801.769,E2 8801.769} C_VEL
LIN {X 0,Y 259.434,Z 455.525,A -85,B 0,C 180,E1 8798.404,E2 8798.404} C_VEL
LIN {X 0,Y 264.142,Z 464.247,A -85,B 0,C 180,E1 8794.915,E2 8794.915} C_VEL
LIN {X 0,Y 267.074,Z 470.47,A -85,B 0,C 180,E1 8792.997,E2 8792.997} C_VEL
LIN {X 0,Y 257.843,Z 579.44,A -85,B 0,C 180,E1 8790.592,E2 8790.592} C_VEL
LIN {X 0,Y 255.589,Z 598.711,A -85,B 0,C 180,E1 8789.912,E2 8789.912} C_VEL
LIN {X 0,Y 252.035,Z 617.628,A -85,B 0,C 180,E1 8788.968,E2 8788.968} C_VEL
LIN {X 0,Y 247.178,Z 636.274,A -85,B 0,C 180,E1 8787.715,E2 8787.715} C_VEL
LIN {X 0,Y 241.308,Z 653.871,A -85,B 0,C 180,E1 8786.175,E2 8786.175} C_VEL
LIN {X 0,Y 234.158,Z 671.292,A -85,B 0,C 180,E1 8784.221,E2 8784.221} C_VEL
LIN {X 0,Y 226.228,Z 687.532,A -85,B 0,C 180,E1 8781.877,E2 8781.877} C_VEL
LIN {X 0,Y 217.745,Z 702.468,A -85,B 0,C 180,E1 8779.116,E2 8779.116} C_VEL
LIN {X 0,Y 208.949,Z 716.095,A -85,B 0,C 180,E1 8775.869,E2 8775.869} C_VEL
LIN {X 0,Y 200.025,Z 728.437,A -85,B 0,C 180,E1 8772.052,E2 8772.052} C_VEL
LIN {X 0,Y 191.434,Z 739.221,A -85,B 0,C 180,E1 8767.667,E2 8767.667} C_VEL
LIN {X 0,Y 183.495,Z 748.46,A -85,B 0,C 180,E1 8762.645,E2 8762.645} C_VEL
LIN {X 0,Y 176.504,Z 756.135,A -85,B 0,C 180,E1 8756.947,E2 8756.947} C_VEL
LIN {X 0,Y 170.775,Z 762.231,A -85,B 0,C 180,E1 8750.481,E2 8750.481} C_VEL
LIN {X 0,Y 166.936,Z 766.334,A -85,B 0,C 180,E1 8743.861,E2 8743.861} C_VEL
LIN {X 0,Y 164.713,Z 768.772,A -85,B 0,C 180,E1 8736.973,E2 8736.973} C_VEL
LIN {X 0,Y 164.019,Z 769.581,A -85,B 0,C 180,E1 8730,E2 8730} C_VEL
LIN {X 0,Y 164.698,Z 768.805,A -85,B 0,C 180,E1 8723.026,E2 8723.026} C_VEL
LIN {X 0,Y 167.009,Z 766.307,A -85,B 0,C 180,E1 8715.902,E2 8715.902} C_VEL
LIN {X 0,Y 171.022,Z 762.045,A -85,B 0,C 180,E1 8709.107,E2 8709.107} C_VEL
LIN {X 0,Y 176.764,Z 755.939,A -85,B 0,C 180,E1 8702.732,E2 8702.732} C_VEL
LIN {X 0,Y 183.818,Z 748.206,A -85,B 0,C 180,E1 8697.049,E2 8697.049} C_VEL
LIN {X 0,Y 191.816,Z 738.903,A -85,B 0,C 180,E1 8692.043,E2 8692.043} C_VEL
LIN {X 0,Y 200.458,Z 728.045,A -85,B 0,C 180,E1 8687.674,E2 8687.674} C_VEL
LIN {X 0,Y 209.421,Z 715.62,A -85,B 0,C 180,E1 8683.87,E2 8683.87} C_VEL
LIN {X 0,Y 218.16,Z 702.06,A -85,B 0,C 180,E1 8680.669,E2 8680.669} C_VEL
LIN {X 0,Y 226.765,Z 686.843,A -85,B 0,C 180,E1 8677.887,E2 8677.887} C_VEL
LIN {X 0,Y 234.719,Z 670.442,A -85,B 0,C 180,E1 8675.551,E2 8675.551} C_VEL
LIN {X 0,Y 241.595,Z 653.631,A -85,B 0,C 180,E1 8673.682,E2 8673.682} C_VEL
LIN {X 0,Y 247.56,Z 635.707,A -85,B 0,C 180,E1 8672.124,E2 8672.124} C_VEL
LIN {X 0,Y 252.462,Z 616.691,A -85,B 0,C 180,E1 8670.863,E2 8670.863} C_VEL
LIN {X 0,Y 256.095,Z 596.836,A -85,B 0,C 180,E1 8669.893,E2 8669.893} C_VEL
LIN {X 0,Y 258.309,Z 576.478,A -85,B 0,C 180,E1 8669.21,E2 8669.21} C_VEL
LIN {X 0,Y 267.24,Z 470.279,A -85,B 0,C 180,E1 8666.858,E2 8666.858} C_VEL
LIN {X 0,Y 262.656,Z 461.236,A -85,B 0,C 180,E1 8663.799,E2 8663.799} C_VEL
LIN {X 0,Y 258.568,Z 454.007,A -85,B 0,C 180,E1 8660.603,E2 8660.603} C_VEL
LIN {X 0,Y 255.072,Z 447.992,A -85,B 0,C 180,E1 8657.215,E2 8657.215} C_VEL
LIN {X 0,Y 252.461,Z 443.849,A -85,B 0,C 180,E1 8653.981,E2 8653.981} C_VEL
LIN {X 0,Y 249.889,Z 439.776,A -85,B 0,C 180,E1 8649.21,E2 8649.21} C_VEL
LIN {X 0,Y 248.64,Z 439.004,A -85,B 0,C 180,E1 8643.459,E2 8643.459} C_VEL
LIN {X 0,Y 249.26,Z 440.065,A -85,B 0,C 180,E1 8638.851,E2 8638.851} C_VEL
LIN {X 0,Y 251.292,Z 444.281,A -85,B 0,C 180,E1 8633.948,E2 8633.948} C_VEL
LIN {X 0,Y 254.152,Z 449.837,A -85,B 0,C 180,E1 8629.918,E2 8629.918} C_VEL
LIN {X 0,Y 257.809,Z 457,A -85,B 0,C 180,E1 8626.144,E2 8626.144} C_VEL
LIN {X 0,Y 261.951,Z 465.547,A -85,B 0,C 180,E1 8622.737,E2 8622.737} C_VEL
LIN {X 0,Y 266.413,Z 475.424,A -85,B 0,C 180,E1 8619.63,E2 8619.63} C_VEL
LIN {X 0,Y 267.328,Z 478.005,A -85,B 0,C 180,E1 8619.015,E2 8619.015} C_VEL
LIN {X 0,Y 264.534,Z 508.324,A -85,B 0,C 180,E1 8618.34,E2 8618.34} C_VEL
LIN {X 0,Y 263.392,Z 516.006,A -85,B 0,C 180,E1 8618.372,E2 8618.372} C_VEL
LIN {X 0,Y 258.909,Z 536.455,A -85,B 0,C 180,E1 8619.164,E2 8619.164} C_VEL
LIN {X 0,Y 257.975,Z 543.047,A -85,B 0,C 180,E1 8619.173,E2 8619.173} C_VEL
LIN {X 0,Y 251.242,Z 612.308,A -85,B 0,C 180,E1 8617.568,E2 8617.568} C_VEL
LIN {X 0,Y 247.509,Z 633.326,A -85,B 0,C 180,E1 8616.872,E2 8616.872} C_VEL
LIN {X 0,Y 242.43,Z 653.082,A -85,B 0,C 180,E1 8615.995,E2 8615.995} C_VEL
LIN {X 0,Y 235.832,Z 672.692,A -85,B 0,C 180,E1 8614.833,E2 8614.833} C_VEL
LIN {X 0,Y 227.817,Z 692.134,A -85,B 0,C 180,E1 8613.266,E2 8613.266} C_VEL
LIN {X 0,Y 218.916,Z 710.457,A -85,B 0,C 180,E1 8611.27,E2 8611.27} C_VEL
LIN {X 0,Y 209.325,Z 727.712,A -85,B 0,C 180,E1 8608.758,E2 8608.758} C_VEL
LIN {X 0,Y 199.25,Z 743.894,A -85,B 0,C 180,E1 8605.635,E2 8605.635} C_VEL
LIN {X 0,Y 188.906,Z 759.069,A -85,B 0,C 180,E1 8601.738,E2 8601.738} C_VEL
LIN {X 0,Y 179.014,Z 772.753,A -85,B 0,C 180,E1 8597.026,E2 8597.026} C_VEL
LIN {X 0,Y 170.232,Z 784.585,A -85,B 0,C 180,E1 8591.581,E2 8591.581} C_VEL
LIN {X 0,Y 162.869,Z 794.852,A -85,B 0,C 180,E1 8585.244,E2 8585.244} C_VEL
LIN {X 0,Y 157.364,Z 803.559,A -85,B 0,C 180,E1 8577.973,E2 8577.973} C_VEL
LIN {X 0,Y 154.381,Z 810.084,A -85,B 0,C 180,E1 8570.47,E2 8570.47} C_VEL
LIN {X 0,Y 153.664,Z 814.529,A -85,B 0,C 180,E1 8563.163,E2 8563.163} C_VEL
LIN {X 0,Y 154.477,Z 817.146,A -85,B 0,C 180,E1 8556.317,E2 8556.317} C_VEL
LIN {X 0,Y 155.33,Z 818.002,A -85,B 0,C 180,E1 8551.475,E2 8551.475} C_VEL
LIN {X 0,Y 155.288,Z 817.963,A -85,B 0,C 180,E1 8548.155,E2 8548.155} C_VEL
LIN {X 0,Y 154.41,Z 817.036,A -85,B 0,C 180,E1 8543.307,E2 8543.307} C_VEL
LIN {X 0,Y 153.66,Z 814.299,A -85,B 0,C 180,E1 8536.453,E2 8536.453} C_VEL
LIN {X 0,Y 154.477,Z 809.738,A -85,B 0,C 180,E1 8529.146,E2 8529.146} C_VEL
LIN {X 0,Y 157.4,Z 803.431,A -85,B 0,C 180,E1 8521.962,E2 8521.962} C_VEL
LIN {X 0,Y 162.907,Z 794.707,A -85,B 0,C 180,E1 8514.715,E2 8514.715} C_VEL
LIN {X 0,Y 170.226,Z 784.474,A -85,B 0,C 180,E1 8508.417,E2 8508.417} C_VEL
LIN {X 0,Y 179.072,Z 772.527,A -85,B 0,C 180,E1 8502.936,E2 8502.936} C_VEL
LIN {X 0,Y 188.874,Z 758.936,A -85,B 0,C 180,E1 8498.27,E2 8498.27} C_VEL
LIN {X 0,Y 198.905,Z 744.208,A -85,B 0,C 180,E1 8494.475,E2 8494.475} C_VEL
LIN {X 0,Y 208.956,Z 728.077,A -85,B 0,C 180,E1 8491.339,E2 8491.339} C_VEL
LIN {X 0,Y 218.658,Z 710.63,A -85,B 0,C 180,E1 8488.784,E2 8488.784} C_VEL
LIN {X 0,Y 227.411,Z 692.631,A -85,B 0,C 180,E1 8486.81,E2 8486.81} C_VEL
LIN {X 0,Y 235.429,Z 673.259,A -85,B 0,C 180,E1 8485.234,E2 8485.234} C_VEL
LIN {X 0,Y 242.213,Z 653.162,A -85,B 0,C 180,E1 8484.035,E2 8484.035} C_VEL
LIN {X 0,Y 247.571,Z 632.171,A -85,B 0,C 180,E1 8483.106,E2 8483.106} C_VEL
LIN {X 0,Y 251.244,Z 610.843,A -85,B 0,C 180,E1 8482.413,E2 8482.413} C_VEL
LIN {X 0,Y 263.553,Z 481.54,A -85,B 0,C 180,E1 8479.473,E2 8479.473} C_VEL
LIN {X 0,Y 259.34,Z 471.766,A -85,B 0,C 180,E1 8476.346,E2 8476.346} C_VEL
LIN {X 0,Y 255.173,Z 462.689,A -85,B 0,C 180,E1 8472.617,E2 8472.617} C_VEL
LIN {X 0,Y 251.911,Z 456.072,A -85,B 0,C 180,E1 8468.904,E2 8468.904} C_VEL
LIN {X 0,Y 249.48,Z 451.09,A -85,B 0,C 180,E1 8465.058,E2 8465.058} C_VEL
LIN {X 0,Y 247.82,Z 447.463,A -85,B 0,C 180,E1 8460.462,E2 8460.462} C_VEL
LIN {X 0,Y 247.462,Z 446.709,A -85,B 0,C 180,E1 8455.132,E2 8455.132} C_VEL
LIN {X 0,Y 248.791,Z 447.765,A -85,B 0,C 180,E1 8450.282,E2 8450.282} C_VEL
LIN {X 0,Y 251.559,Z 452.405,A -85,B 0,C 180,E1 8445.381,E2 8445.381} C_VEL
LIN {X 0,Y 254.284,Z 457.06,A -85,B 0,C 180,E1 8442.139,E2 8442.139} C_VEL
LIN {X 0,Y 257.727,Z 463.073,A -85,B 0,C 180,E1 8438.91,E2 8438.91} C_VEL
LIN {X 0,Y 261.996,Z 471.32,A -85,B 0,C 180,E1 8435.599,E2 8435.599} C_VEL
LIN {X 0,Y 263.551,Z 474.897,A -85,B 0,C 180,E1 8434.498,E2 8434.498} C_VEL
LIN {X 0,Y 254.321,Z 580.204,A -85,B 0,C 180,E1 8432.19,E2 8432.19} C_VEL
LIN {X 0,Y 251.971,Z 599.566,A -85,B 0,C 180,E1 8431.512,E2 8431.512} C_VEL
LIN {X 0,Y 248.294,Z 618.521,A -85,B 0,C 180,E1 8430.574,E2 8430.574} C_VEL
LIN {X 0,Y 243.3,Z 637.125,A -85,B 0,C 180,E1 8429.339,E2 8429.339} C_VEL
LIN {X 0,Y 237.016,Z 655.319,A -85,B 0,C 180,E1 8427.757,E2 8427.757} C_VEL
LIN {X 0,Y 229.638,Z 672.656,A -85,B 0,C 180,E1 8425.817,E2 8425.817} C_VEL
LIN {X 0,Y 221.442,Z 688.842,A -85,B 0,C 180,E1 8423.483,E2 8423.483} C_VEL
LIN {X 0,Y 212.56,Z 703.893,A -85,B 0,C 180,E1 8420.694,E2 8420.694} C_VEL
LIN {X 0,Y 203.521,Z 717.348,A -85,B 0,C 180,E1 8417.468,E2 8417.468} C_VEL
LIN {X 0,Y 194.218,Z 729.672,A -85,B 0,C 180,E1 8413.617,E2 8413.617} C_VEL
LIN {X 0,Y 185.224,Z 740.445,A -85,B 0,C 180,E1 8409.165,E2 8409.165} C_VEL
LIN {X 0,Y 176.868,Z 749.676,A -85,B 0,C 180,E1 8404.031,E2 8404.031} C_VEL
LIN {X 0,Y 169.47,Z 757.345,A -85,B 0,C 180,E1 8398.163,E2 8398.163} C_VEL
LIN {X 0,Y 163.427,Z 763.382,A -85,B 0,C 180,E1 8391.535,E2 8391.535} C_VEL
LIN {X 0,Y 159.252,Z 767.538,A -85,B 0,C 180,E1 8384.544,E2 8384.544} C_VEL
LIN {X 0,Y 156.86,Z 769.974,A -85,B 0,C 180,E1 8377.324,E2 8377.324} C_VEL
LIN {X 0,Y 156.11,Z 770.782,A -85,B 0,C 180,E1 8370,E2 8370} C_VEL
LIN {X 0,Y 156.844,Z 770.007,A -85,B 0,C 180,E1 8362.675,E2 8362.675} C_VEL
LIN {X 0,Y 159.218,Z 767.61,A -85,B 0,C 180,E1 8355.452,E2 8355.452} C_VEL
LIN {X 0,Y 163.375,Z 763.49,A -85,B 0,C 180,E1 8348.458,E2 8348.458} C_VEL
LIN {X 0,Y 169.4,Z 757.502,A -85,B 0,C 180,E1 8341.825,E2 8341.825} C_VEL
LIN {X 0,Y 176.785,Z 749.885,A -85,B 0,C 180,E1 8335.951,E2 8335.951} C_VEL
LIN {X 0,Y 185.13,Z 740.702,A -85,B 0,C 180,E1 8330.811,E2 8330.811} C_VEL
LIN {X 0,Y 194.118,Z 729.979,A -85,B 0,C 180,E1 8326.355,E2 8326.355} C_VEL
LIN {X 0,Y 203.414,Z 717.718,A -85,B 0,C 180,E1 8322.499,E2 8322.499} C_VEL
LIN {X 0,Y 212.774,Z 703.843,A -85,B 0,C 180,E1 8319.164,E2 8319.164} C_VEL
LIN {X 0,Y 221.669,Z 688.775,A -85,B 0,C 180,E1 8316.379,E2 8316.379} C_VEL
LIN {X 0,Y 229.879,Z 672.569,A -85,B 0,C 180,E1 8314.049,E2 8314.049} C_VEL
LIN {X 0,Y 237.266,Z 655.21,A -85,B 0,C 180,E1 8312.113,E2 8312.113} C_VEL
LIN {X 0,Y 243.69,Z 636.573,A -85,B 0,C 180,E1 8310.503,E2 8310.503} C_VEL
LIN {X 0,Y 248.705,Z 617.715,A -85,B 0,C 180,E1 8309.265,E2 8309.265} C_VEL
LIN {X 0,Y 252.48,Z 597.798,A -85,B 0,C 180,E1 8308.299,E2 8308.299} C_VEL
LIN {X 0,Y 254.79,Z 577.427,A -85,B 0,C 180,E1 8307.618,E2 8307.618} C_VEL
LIN {X 0,Y 263.739,Z 474.717,A -85,B 0,C 180,E1 8305.366,E2 8305.366} C_VEL
LIN {X 0,Y 259.552,Z 466.229,A -85,B 0,C 180,E1 8302.3,E2 8302.3} C_VEL
LIN {X 0,Y 255.458,Z 458.844,A -85,B 0,C 180,E1 8298.71,E2 8298.71} C_VEL
LIN {X 0,Y 252.926,Z 454.585,A -85,B 0,C 180,E1 8295.947,E2 8295.947} C_VEL
LIN {X 0,Y 251.182,Z 451.572,A -85,B 0,C 180,E1 8293.584,E2 8293.584} C_VEL
LIN {X 0,Y 248.738,Z 447.601,A -85,B 0,C 180,E1 8288.787,E2 8288.787} C_VEL
LIN {X 0,Y 247.663,Z 446.989,A -85,B 0,C 180,E1 8283.009,E2 8283.009} C_VEL
LIN {X 0,Y 248.204,Z 447.955,A -85,B 0,C 180,E1 8279.077,E2 8279.077} C_VEL
LIN {X 0,Y 250.085,Z 452.118,A -85,B 0,C 180,E1 8274.264,E2 8274.264} C_VEL
LIN {X 0,Y 252.656,Z 457.359,A -85,B 0,C 180,E1 8270.433,E2 8270.433} C_VEL
LIN {X 0,Y 256.105,Z 464.467,A -85,B 0,C 180,E1 8266.683,E2 8266.683} C_VEL
LIN {X 0,Y 260.086,Z 473.128,A -85,B 0,C 180,E1 8263.243,E2 8263.243} C_VEL
LIN {X 0,Y 263.781,Z 481.757,A -85,B 0,C 180,E1 8260.523,E2 8260.523} C_VEL
LIN {X 0,Y 257.975,Z 543.047,A -85,B 0,C 180,E1 8259.173,E2 8259.173} C_VEL
LIN {X 0,Y 256.837,Z 550.729,A -85,B 0,C 180,E1 8259.207,E2 8259.207} C_VEL
LIN {X 0,Y 252.404,Z 571.175,A -85,B 0,C 180,E1 8260.036,E2 8260.036} C_VEL
LIN {X 0,Y 251.472,Z 577.768,A -85,B 0,C 180,E1 8260.05,E2 8260.05} C_VEL
LIN {X 0,Y 247.799,Z 612.659,A -85,B 0,C 180,E1 8259.224,E2 8259.224} C_VEL
LIN {X 0,Y 244.011,Z 633.123,A -85,B 0,C 180,E1 8258.555,E2 8258.555} C_VEL
LIN {X 0,Y 238.821,Z 652.717,A -85,B 0,C 180,E1 8257.702,E2 8257.702} C_VEL
LIN {X 0,Y 232.091,Z 672.178,A -85,B 0,C 180,E1 8256.576,E2 8256.576} C_VEL
LIN {X 0,Y 223.86,Z 691.55,A -85,B 0,C 180,E1 8255.048,E2 8255.048} C_VEL
LIN {X 0,Y 214.706,Z 709.79,A -85,B 0,C 180,E1 8253.096,E2 8253.096} C_VEL
LIN {X 0,Y 204.803,Z 726.974,A -85,B 0,C 180,E1 8250.624,E2 8250.624} C_VEL
LIN {X 0,Y 194.35,Z 743.09,A -85,B 0,C 180,E1 8247.532,E2 8247.532} C_VEL
LIN {X 0,Y 183.658,Z 758.072,A -85,B 0,C 180,E1 8243.679,E2 8243.679} C_VEL
LIN {X 0,Y 173.438,Z 771.461,A -85,B 0,C 180,E1 8239.041,E2 8239.041} C_VEL
LIN {X 0,Y 164.084,Z 783.3,A -85,B 0,C 180,E1 8233.516,E2 8233.516} C_VEL
LIN {X 0,Y 156.127,Z 793.575,A -85,B 0,C 180,E1 8227.011,E2 8227.011} C_VEL
LIN {X 0,Y 150.1,Z 802.221,A -85,B 0,C 180,E1 8219.533,E2 8219.533} C_VEL
LIN {X 0,Y 146.653,Z 808.825,A -85,B 0,C 180,E1 8211.602,E2 8211.602} C_VEL
LIN {X 0,Y 145.702,Z 813.285,A -85,B 0,C 180,E1 8203.897,E2 8203.897} C_VEL
LIN {X 0,Y 146.466,Z 815.921,A -85,B 0,C 180,E1 8196.664,E2 8196.664} C_VEL
LIN {X 0,Y 147.401,Z 816.797,A -85,B 0,C 180,E1 8191.555,E2 8191.555} C_VEL
LIN {X 0,Y 147.351,Z 816.757,A -85,B 0,C 180,E1 8188.056,E2 8188.056} C_VEL
LIN {X 0,Y 146.324,Z 815.709,A -85,B 0,C 180,E1 8182.54,E2 8182.54} C_VEL
LIN {X 0,Y 145.711,Z 812.851,A -85,B 0,C 180,E1 8175.292,E2 8175.292} C_VEL
LIN {X 0,Y 147.013,Z 807.873,A -85,B 0,C 180,E1 8167.191,E2 8167.191} C_VEL
LIN {X 0,Y 150.608,Z 801.312,A -85,B 0,C 180,E1 8159.659,E2 8159.659} C_VEL
LIN {X 0,Y 156.491,Z 792.975,A -85,B 0,C 180,E1 8152.63,E2 8152.63} C_VEL
LIN {X 0,Y 164.082,Z 783.179,A -85,B 0,C 180,E1 8146.48,E2 8146.48} C_VEL
LIN {X 0,Y 173.432,Z 771.32,A -85,B 0,C 180,E1 8140.956,E2 8140.956} C_VEL
LIN {X 0,Y 183.65,Z 757.9,A -85,B 0,C 180,E1 8136.318,E2 8136.318} C_VEL
LIN {X 0,Y 194.34,Z 742.872,A -85,B 0,C 180,E1 8132.463,E2 8132.463} C_VEL
LIN {X 0,Y 204.792,Z 726.711,A -85,B 0,C 180,E1 8129.37,E2 8129.37} C_VEL
LIN {X 0,Y 214.696,Z 709.474,A -85,B 0,C 180,E1 8126.899,E2 8126.899} C_VEL
LIN {X 0,Y 223.85,Z 691.159,A -85,B 0,C 180,E1 8124.946,E2 8124.946} C_VEL
LIN {X 0,Y 231.87,Z 672.23,A -85,B 0,C 180,E1 8123.455,E2 8123.455} C_VEL
LIN {X 0,Y 238.81,Z 652.104,A -85,B 0,C 180,E1 8122.292,E2 8122.292} C_VEL
LIN {X 0,Y 244.27,Z 631.118,A -85,B 0,C 180,E1 8121.391,E2 8121.391} C_VEL
LIN {X 0,Y 248,Z 609.891,A -85,B 0,C 180,E1 8120.719,E2 8120.719} C_VEL
LIN {X 0,Y 260.144,Z 485.777,A -85,B 0,C 180,E1 8117.938,E2 8117.938} C_VEL
LIN {X 0,Y 256.385,Z 476.76,A -85,B 0,C 180,E1 8114.857,E2 8114.857} C_VEL
LIN {X 0,Y 252.994,Z 469.085,A -85,B 0,C 180,E1 8111.512,E2 8111.512} C_VEL
LIN {X 0,Y 250.154,Z 462.889,A -85,B 0,C 180,E1 8107.926,E2 8107.926} C_VEL
LIN {X 0,Y 248.129,Z 458.615,A -85,B 0,C 180,E1 8104.391,E2 8104.391} C_VEL
LIN {X 0,Y 246.784,Z 455.352,A -85,B 0,C 180,E1 8100.232,E2 8100.232} C_VEL
LIN {X 0,Y 246.49,Z 454.651,A -85,B 0,C 180,E1 8095.113,E2 8095.113} C_VEL
LIN {X 0,Y 247.721,Z 455.697,A -85,B 0,C 180,E1 8090.474,E2 8090.474} C_VEL
LIN {X 0,Y 250.266,Z 460.124,A -85,B 0,C 180,E1 8085.776,E2 8085.776} C_VEL
LIN {X 0,Y 252.789,Z 464.632,A -85,B 0,C 180,E1 8082.624,E2 8082.624} C_VEL
LIN {X 0,Y 256.044,Z 470.619,A -85,B 0,C 180,E1 8079.423,E2 8079.423} C_VEL
LIN {X 0,Y 259.951,Z 478.537,A -85,B 0,C 180,E1 8076.244,E2 8076.244} C_VEL
LIN {X 0,Y 260.188,Z 479.476,A -85,B 0,C 180,E1 8076.034,E2 8076.034} C_VEL
LIN {X 0,Y 251.001,Z 580.966,A -85,B 0,C 180,E1 8073.832,E2 8073.832} C_VEL
LIN {X 0,Y 248.557,Z 600.417,A -85,B 0,C 180,E1 8073.157,E2 8073.157} C_VEL
LIN {X 0,Y 244.717,Z 619.559,A -85,B 0,C 180,E1 8072.221,E2 8072.221} C_VEL
LIN {X 0,Y 239.517,Z 638.294,A -85,B 0,C 180,E1 8070.989,E2 8070.989} C_VEL
LIN {X 0,Y 233.278,Z 655.875,A -85,B 0,C 180,E1 8069.484,E2 8069.484} C_VEL
LIN {X 0,Y 225.771,Z 673.077,A -85,B 0,C 180,E1 8067.597,E2 8067.597} C_VEL
LIN {X 0,Y 217.188,Z 689.557,A -85,B 0,C 180,E1 8065.258,E2 8065.258} C_VEL
LIN {X 0,Y 207.98,Z 704.672,A -85,B 0,C 180,E1 8062.487,E2 8062.487} C_VEL
LIN {X 0,Y 198.259,Z 718.598,A -85,B 0,C 180,E1 8059.153,E2 8059.153} C_VEL
LIN {X 0,Y 188.564,Z 730.905,A -85,B 0,C 180,E1 8055.277,E2 8055.277} C_VEL
LIN {X 0,Y 179.149,Z 741.668,A -85,B 0,C 180,E1 8050.766,E2 8050.766} C_VEL
LIN {X 0,Y 170.352,Z 750.892,A -85,B 0,C 180,E1 8045.525,E2 8045.525} C_VEL
LIN {X 0,Y 162.518,Z 758.555,A -85,B 0,C 180,E1 8039.483,E2 8039.483} C_VEL
LIN {X 0,Y 156.075,Z 764.587,A -85,B 0,C 180,E1 8032.604,E2 8032.604} C_VEL
LIN {X 0,Y 151.594,Z 768.742,A -85,B 0,C 180,E1 8025.297,E2 8025.297} C_VEL
LIN {X 0,Y 149.013,Z 771.177,A -85,B 0,C 180,E1 8017.712,E2 8017.712} C_VEL
LIN {X 0,Y 148.201,Z 771.984,A -85,B 0,C 180,E1 8010,E2 8010} C_VEL
LIN {X 0,Y 148.996,Z 771.208,A -85,B 0,C 180,E1 8002.287,E2 8002.287} C_VEL
LIN {X 0,Y 151.559,Z 768.813,A -85,B 0,C 180,E1 7994.7,E2 7994.7} C_VEL
LIN {X 0,Y 156.133,Z 764.602,A -85,B 0,C 180,E1 7987.246,E2 7987.246} C_VEL
LIN {X 0,Y 162.449,Z 758.708,A -85,B 0,C 180,E1 7980.503,E2 7980.503} C_VEL
LIN {X 0,Y 170.27,Z 751.095,A -85,B 0,C 180,E1 7974.456,E2 7974.456} C_VEL
LIN {X 0,Y 179.056,Z 741.918,A -85,B 0,C 180,E1 7969.208,E2 7969.208} C_VEL
LIN {X 0,Y 188.466,Z 731.205,A -85,B 0,C 180,E1 7964.693,E2 7964.693} C_VEL
LIN {X 0,Y 198.154,Z 718.96,A -85,B 0,C 180,E1 7960.812,E2 7960.812} C_VEL
LIN {X 0,Y 207.872,Z 705.108,A -85,B 0,C 180,E1 7957.475,E2 7957.475} C_VEL
LIN {X 0,Y 217.158,Z 689.944,A -85,B 0,C 180,E1 7954.679,E2 7954.679} C_VEL
LIN {X 0,Y 225.558,Z 673.92,A -85,B 0,C 180,E1 7952.39,E2 7952.39} C_VEL
LIN {X 0,Y 233.175,Z 656.639,A -85,B 0,C 180,E1 7950.473,E2 7950.473} C_VEL
LIN {X 0,Y 239.573,Z 638.784,A -85,B 0,C 180,E1 7948.934,E2 7948.934} C_VEL
LIN {X 0,Y 244.673,Z 620.585,A -85,B 0,C 180,E1 7947.727,E2 7947.727} C_VEL
LIN {X 0,Y 248.553,Z 601.667,A -85,B 0,C 180,E1 7946.784,E2 7946.784} C_VEL
LIN {X 0,Y 251.088,Z 582.292,A -85,B 0,C 180,E1 7946.096,E2 7946.096} C_VEL
LIN {X 0,Y 257.593,Z 510.007,A -85,B 0,C 180,E1 7944.486,E2 7944.486} C_VEL
LIN {X 0,Y 260.403,Z 479.233,A -85,B 0,C 180,E1 7943.831,E2 7943.831} C_VEL
LIN {X 0,Y 256.523,Z 471.34,A -85,B 0,C 180,E1 7940.702,E2 7940.702} C_VEL
LIN {X 0,Y 253.207,Z 465.166,A -85,B 0,C 180,E1 7937.465,E2 7937.465} C_VEL
LIN {X 0,Y 251.234,Z 461.709,A -85,B 0,C 180,E1 7935.111,E2 7935.111} C_VEL
LIN {X 0,Y 249.755,Z 459.117,A -85,B 0,C 180,E1 7932.956,E2 7932.956} C_VEL
LIN {X 0,Y 247.684,Z 455.499,A -85,B 0,C 180,E1 7928.591,E2 7928.591} C_VEL
LIN {X 0,Y 246.69,Z 454.93,A -85,B 0,C 180,E1 7923.021,E2 7923.021} C_VEL
LIN {X 0,Y 247.153,Z 455.842,A -85,B 0,C 180,E1 7919.305,E2 7919.305} C_VEL
LIN {X 0,Y 248.83,Z 459.798,A -85,B 0,C 180,E1 7914.698,E2 7914.698} C_VEL
LIN {X 0,Y 251.269,Z 465.053,A -85,B 0,C 180,E1 7910.842,E2 7910.842} C_VEL
LIN {X 0,Y 254.479,Z 472.046,A -85,B 0,C 180,E1 7907.174,E2 7907.174} C_VEL
LIN {X 0,Y 258.364,Z 481.072,A -85,B 0,C 180,E1 7903.648,E2 7903.648} C_VEL
LIN {X 0,Y 260.366,Z 486.215,A -85,B 0,C 180,E1 7902.046,E2 7902.046} C_VEL
LIN {X 0,Y 251.472,Z 577.768,A -85,B 0,C 180,E1 7900.05,E2 7900.05} C_VEL
LIN {X 0,Y 250.377,Z 585.457,A -85,B 0,C 180,E1 7900.094,E2 7900.094} C_VEL
LIN {X 0,Y 245.903,Z 605.889,A -85,B 0,C 180,E1 7900.952,E2 7900.952} C_VEL
LIN {X 0,Y 244.663,Z 612.431,A -85,B 0,C 180,E1 7900.942,E2 7900.942} C_VEL
LIN {X 0,Y 240.783,Z 632.702,A -85,B 0,C 180,E1 7900.293,E2 7900.293} C_VEL
LIN {X 0,Y 235.429,Z 652.333,A -85,B 0,C 180,E1 7899.46,E2 7899.46} C_VEL
LIN {X 0,Y 228.669,Z 671.403,A -85,B 0,C 180,E1 7898.391,E2 7898.391} C_VEL
LIN {X 0,Y 220.544,Z 690.09,A -85,B 0,C 180,E1 7896.969,E2 7896.969} C_VEL
LIN {X 0,Y 211.054,Z 708.526,A -85,B 0,C 180,E1 7895.063,E2 7895.063} C_VEL
LIN {X 0,Y 200.748,Z 725.851,A -85,B 0,C 180,E1 7892.634,E2 7892.634} C_VEL
LIN {X 0,Y 189.676,Z 742.276,A -85,B 0,C 180,E1 7889.525,E2 7889.525} C_VEL
LIN {X 0,Y 178.87,Z 756.768,A -85,B 0,C 180,E1 7885.82,E2 7885.82} C_VEL
LIN {X 0,Y 168.095,Z 770.168,A -85,B 0,C 180,E1 7881.186,E2 7881.186} C_VEL
LIN {X 0,Y 158.139,Z 782.016,A -85,B 0,C 180,E1 7875.597,E2 7875.597} C_VEL
LIN {X 0,Y 149.543,Z 792.296,A -85,B 0,C 180,E1 7868.938,E2 7868.938} C_VEL
LIN {X 0,Y 142.909,Z 800.951,A -85,B 0,C 180,E1 7861.179,E2 7861.179} C_VEL
LIN {X 0,Y 138.985,Z 807.564,A -85,B 0,C 180,E1 7852.859,E2 7852.859} C_VEL
LIN {X 0,Y 137.753,Z 812.039,A -85,B 0,C 180,E1 7844.716,E2 7844.716} C_VEL
LIN {X 0,Y 138.445,Z 814.695,A -85,B 0,C 180,E1 7837.052,E2 7837.052} C_VEL
LIN {X 0,Y 139.466,Z 815.591,A -85,B 0,C 180,E1 7831.643,E2 7831.643} C_VEL
LIN {X 0,Y 139.466,Z 815.586,A -85,B 0,C 180,E1 7828.357,E2 7828.357} C_VEL
LIN {X 0,Y 138.448,Z 814.681,A -85,B 0,C 180,E1 7822.948,E2 7822.948} C_VEL
LIN {X 0,Y 137.765,Z 811.803,A -85,B 0,C 180,E1 7814.853,E2 7814.853} C_VEL
LIN {X 0,Y 139.121,Z 807.214,A -85,B 0,C 180,E1 7806.717,E2 7806.717} C_VEL
LIN {X 0,Y 142.907,Z 800.885,A -85,B 0,C 180,E1 7798.82,E2 7798.82} C_VEL
LIN {X 0,Y 149.54,Z 792.205,A -85,B 0,C 180,E1 7791.061,E2 7791.061} C_VEL
LIN {X 0,Y 158.135,Z 781.896,A -85,B 0,C 180,E1 7784.401,E2 7784.401} C_VEL
LIN {X 0,Y 168.089,Z 770.02,A -85,B 0,C 180,E1 7778.811,E2 7778.811} C_VEL
LIN {X 0,Y 178.861,Z 756.587,A -85,B 0,C 180,E1 7774.176,E2 7774.176} C_VEL
LIN {X 0,Y 190.029,Z 741.535,A -85,B 0,C 180,E1 7770.358,E2 7770.358} C_VEL
LIN {X 0,Y 200.882,Z 725.341,A -85,B 0,C 180,E1 7767.323,E2 7767.323} C_VEL
LIN {X 0,Y 210.959,Z 708.352,A -85,B 0,C 180,E1 7764.949,E2 7764.949} C_VEL
LIN {X 0,Y 220.118,Z 690.564,A -85,B 0,C 180,E1 7763.102,E2 7763.102} C_VEL
LIN {X 0,Y 228.119,Z 672.224,A -85,B 0,C 180,E1 7761.692,E2 7761.692} C_VEL
LIN {X 0,Y 234.988,Z 653.026,A -85,B 0,C 180,E1 7760.6,E2 7760.6} C_VEL
LIN {X 0,Y 240.448,Z 633.199,A -85,B 0,C 180,E1 7759.749,E2 7759.749} C_VEL
LIN {X 0,Y 244.372,Z 612.887,A -85,B 0,C 180,E1 7759.092,E2 7759.092} C_VEL
LIN {X 0,Y 247.847,Z 581.803,A -85,B 0,C 180,E1 7758.357,E2 7758.357} C_VEL
LIN {X 0,Y 256.947,Z 490.156,A -85,B 0,C 180,E1 7756.386,E2 7756.386} C_VEL
LIN {X 0,Y 253.38,Z 481.296,A -85,B 0,C 180,E1 7753.114,E2 7753.114} C_VEL
LIN {X 0,Y 250.863,Z 475.413,A -85,B 0,C 180,E1 7750.332,E2 7750.332} C_VEL
LIN {X 0,Y 248.668,Z 470.294,A -85,B 0,C 180,E1 7747.276,E2 7747.276} C_VEL
LIN {X 0,Y 246.914,Z 466.316,A -85,B 0,C 180,E1 7743.947,E2 7743.947} C_VEL
LIN {X 0,Y 245.743,Z 463.239,A -85,B 0,C 180,E1 7740,E2 7740} C_VEL
LIN {X 0,Y 245.547,Z 462.608,A -85,B 0,C 180,E1 7734.86,E2 7734.86} C_VEL
LIN {X 0,Y 246.654,Z 463.625,A -85,B 0,C 180,E1 7730.668,E2 7730.668} C_VEL
LIN {X 0,Y 248.984,Z 467.843,A -85,B 0,C 180,E1 7726.176,E2 7726.176} C_VEL
LIN {X 0,Y 251.404,Z 472.39,A -85,B 0,C 180,E1 7723.003,E2 7723.003} C_VEL
LIN {X 0,Y 254.563,Z 478.529,A -85,B 0,C 180,E1 7719.779,E2 7719.779} C_VEL
LIN {X 0,Y 257.045,Z 483.834,A -85,B 0,C 180,E1 7717.615,E2 7717.615} C_VEL
LIN {X 0,Y 247.915,Z 581.507,A -85,B 0,C 180,E1 7715.523,E2 7715.523} C_VEL
LIN {X 0,Y 245.389,Z 601.071,A -85,B 0,C 180,E1 7714.855,E2 7714.855} C_VEL
LIN {X 0,Y 241.502,Z 620.015,A -85,B 0,C 180,E1 7713.947,E2 7713.947} C_VEL
LIN {X 0,Y 236.186,Z 638.749,A -85,B 0,C 180,E1 7712.745,E2 7712.745} C_VEL
LIN {X 0,Y 229.38,Z 657.321,A -85,B 0,C 180,E1 7711.179,E2 7711.179} C_VEL
LIN {X 0,Y 221.535,Z 674.663,A -85,B 0,C 180,E1 7709.29,E2 7709.29} C_VEL
LIN {X 0,Y 212.789,Z 690.868,A -85,B 0,C 180,E1 7707.005,E2 7707.005} C_VEL
LIN {X 0,Y 203.265,Z 705.946,A -85,B 0,C 180,E1 7704.254,E2 7704.254} C_VEL
LIN {X 0,Y 193.177,Z 719.844,A -85,B 0,C 180,E1 7700.928,E2 7700.928} C_VEL
LIN {X 0,Y 183.078,Z 732.135,A -85,B 0,C 180,E1 7697.038,E2 7697.038} C_VEL
LIN {X 0,Y 173.224,Z 742.889,A -85,B 0,C 180,E1 7692.478,E2 7692.478} C_VEL
LIN {X 0,Y 163.96,Z 752.107,A -85,B 0,C 180,E1 7687.136,E2 7687.136} C_VEL
LIN {X 0,Y 155.661,Z 759.765,A -85,B 0,C 180,E1 7680.921,E2 7680.921} C_VEL
LIN {X 0,Y 148.783,Z 765.793,A -85,B 0,C 180,E1 7673.779,E2 7673.779} C_VEL
LIN {X 0,Y 143.964,Z 769.946,A -85,B 0,C 180,E1 7666.129,E2 7666.129} C_VEL
LIN {X 0,Y 141.173,Z 772.379,A -85,B 0,C 180,E1 7658.143,E2 7658.143} C_VEL
LIN {X 0,Y 140.292,Z 773.185,A -85,B 0,C 180,E1 7650,E2 7650} C_VEL
LIN {X 0,Y 141.156,Z 772.41,A -85,B 0,C 180,E1 7641.856,E2 7641.856} C_VEL
LIN {X 0,Y 143.929,Z 770.016,A -85,B 0,C 180,E1 7633.867,E2 7633.867} C_VEL
LIN {X 0,Y 148.729,Z 765.899,A -85,B 0,C 180,E1 7626.212,E2 7626.212} C_VEL
LIN {X 0,Y 155.591,Z 759.914,A -85,B 0,C 180,E1 7619.064,E2 7619.064} C_VEL
LIN {X 0,Y 163.879,Z 752.305,A -85,B 0,C 180,E1 7612.843,E2 7612.843} C_VEL
LIN {X 0,Y 173.131,Z 743.134,A -85,B 0,C 180,E1 7607.494,E2 7607.494} C_VEL
LIN {X 0,Y 182.982,Z 732.43,A -85,B 0,C 180,E1 7602.93,E2 7602.93} C_VEL
LIN {X 0,Y 193.075,Z 720.2,A -85,B 0,C 180,E1 7599.035,E2 7599.035} C_VEL
LIN {X 0,Y 203.161,Z 706.372,A -85,B 0,C 180,E1 7595.706,E2 7595.706} C_VEL
LIN {X 0,Y 212.685,Z 691.374,A -85,B 0,C 180,E1 7592.952,E2 7592.952} C_VEL
LIN {X 0,Y 221.287,Z 675.555,A -85,B 0,C 180,E1 7590.703,E2 7590.703} C_VEL
LIN {X 0,Y 228.902,Z 658.944,A -85,B 0,C 180,E1 7588.864,E2 7588.864} C_VEL
LIN {X 0,Y 235.329,Z 641.891,A -85,B 0,C 180,E1 7587.381,E2 7587.381} C_VEL
LIN {X 0,Y 240.875,Z 623.254,A -85,B 0,C 180,E1 7586.128,E2 7586.128} C_VEL
LIN {X 0,Y 245.108,Z 603.844,A -85,B 0,C 180,E1 7585.152,E2 7585.152} C_VEL
LIN {X 0,Y 247.888,Z 583.957,A -85,B 0,C 180,E1 7584.438,E2 7584.438} C_VEL
LIN {X 0,Y 253.751,Z 520.881,A -85,B 0,C 180,E1 7583.031,E2 7583.031} C_VEL
LIN {X 0,Y 257.195,Z 483.763,A -85,B 0,C 180,E1 7582.224,E2 7582.224} C_VEL
LIN {X 0,Y 253.712,Z 476.578,A -85,B 0,C 180,E1 7579.093,E2 7579.093} C_VEL
LIN {X 0,Y 250.608,Z 470.559,A -85,B 0,C 180,E1 7575.624,E2 7575.624} C_VEL
LIN {X 0,Y 248.499,Z 466.835,A -85,B 0,C 180,E1 7572.549,E2 7572.549} C_VEL
LIN {X 0,Y 246.632,Z 463.397,A -85,B 0,C 180,E1 7568.393,E2 7568.393} C_VEL
LIN {X 0,Y 245.708,Z 462.87,A -85,B 0,C 180,E1 7563.033,E2 7563.033} C_VEL
LIN {X 0,Y 246.106,Z 463.728,A -85,B 0,C 180,E1 7559.535,E2 7559.535} C_VEL
LIN {X 0,Y 247.641,Z 467.633,A -85,B 0,C 180,E1 7555.021,E2 7555.021} C_VEL
LIN {X 0,Y 249.902,Z 472.748,A -85,B 0,C 180,E1 7551.255,E2 7551.255} C_VEL
LIN {X 0,Y 252.815,Z 479.538,A -85,B 0,C 180,E1 7547.727,E2 7547.727} C_VEL
LIN {X 0,Y 256.4,Z 488.415,A -85,B 0,C 180,E1 7544.275,E2 7544.275} C_VEL
LIN {X 0,Y 257.139,Z 490.654,A -85,B 0,C 180,E1 7543.613,E2 7543.613} C_VEL
LIN {X 0,Y 245.047,Z 610.055,A -85,B 0,C 180,E1 7541.01,E2 7541.01} C_VEL
LIN {X 0,Y 244.663,Z 612.431,A -85,B 0,C 180,E1 7540.942,E2 7540.942} C_VEL
LIN {X 0,Y 243.006,Z 620.009,A -85,B 0,C 180,E1 7540.97,E2 7540.97} C_VEL
LIN {X 0,Y 236.841,Z 637.813,A -85,B 0,C 180,E1 7541.609,E2 7541.609} C_VEL
LIN {X 0,Y 234.337,Z 645.192,A -85,B 0,C 180,E1 7541.564,E2 7541.564} C_VEL
LIN {X 0,Y 234.022,Z 646.228,A -85,B 0,C 180,E1 7541.524,E2 7541.524} C_VEL
LIN {X 0,Y 227.43,Z 665.555,A -85,B 0,C 180,E1 7540.559,E2 7540.559} C_VEL
LIN {X 0,Y 219.189,Z 684.926,A -85,B 0,C 180,E1 7539.245,E2 7539.245} C_VEL
LIN {X 0,Y 209.883,Z 703.202,A -85,B 0,C 180,E1 7537.543,E2 7537.543} C_VEL
LIN {X 0,Y 199.515,Z 720.678,A -85,B 0,C 180,E1 7535.33,E2 7535.33} C_VEL
LIN {X 0,Y 188.277,Z 737.25,A -85,B 0,C 180,E1 7532.478,E2 7532.478} C_VEL
LIN {X 0,Y 177.173,Z 751.883,A -85,B 0,C 180,E1 7529.067,E2 7529.067} C_VEL
LIN {X 0,Y 166.211,Z 765.114,A -85,B 0,C 180,E1 7524.895,E2 7524.895} C_VEL
LIN {X 0,Y 155.772,Z 776.983,A -85,B 0,C 180,E1 7519.801,E2 7519.801} C_VEL
LIN {X 0,Y 146.309,Z 787.449,A -85,B 0,C 180,E1 7513.646,E2 7513.646} C_VEL
LIN {X 0,Y 138.442,Z 796.451,A -85,B 0,C 180,E1 7506.314,E2 7506.314} C_VEL
LIN {X 0,Y 133.041,Z 803.577,A -85,B 0,C 180,E1 7498.259,E2 7498.259} C_VEL
LIN {X 0,Y 130.135,Z 809.242,A -85,B 0,C 180,E1 7489.087,E2 7489.087} C_VEL
LIN {X 0,Y 129.976,Z 812.621,A -85,B 0,C 180,E1 7480.639,E2 7480.639} C_VEL
LIN {X 0,Y 131.211,Z 814.223,A -85,B 0,C 180,E1 7473.402,E2 7473.402} C_VEL
LIN {X 0,Y 131.671,Z 814.48,A -85,B 0,C 180,E1 7469.565,E2 7469.565} C_VEL
LIN {X 0,Y 130.744,Z 813.85,A -85,B 0,C 180,E1 7464.294,E2 7464.294} C_VEL
LIN {X 0,Y 129.807,Z 811.681,A -85,B 0,C 180,E1 7456.64,E2 7456.64} C_VEL
LIN {X 0,Y 130.727,Z 807.581,A -85,B 0,C 180,E1 7447.99,E2 7447.99} C_VEL
LIN {X 0,Y 134.463,Z 801.416,A -85,B 0,C 180,E1 7439.132,E2 7439.132} C_VEL
LIN {X 0,Y 140.678,Z 793.709,A -85,B 0,C 180,E1 7431.286,E2 7431.286} C_VEL
LIN {X 0,Y 149.409,Z 783.877,A -85,B 0,C 180,E1 7424.104,E2 7424.104} C_VEL
LIN {X 0,Y 159.903,Z 772.197,A -85,B 0,C 180,E1 7418.016,E2 7418.016} C_VEL
LIN {X 0,Y 170.874,Z 759.42,A -85,B 0,C 180,E1 7413.203,E2 7413.203} C_VEL
LIN {X 0,Y 182.255,Z 745.141,A -85,B 0,C 180,E1 7409.278,E2 7409.278} C_VEL
LIN {X 0,Y 193.273,Z 729.866,A -85,B 0,C 180,E1 7406.181,E2 7406.181} C_VEL
LIN {X 0,Y 203.564,Z 713.828,A -85,B 0,C 180,E1 7403.751,E2 7403.751} C_VEL
LIN {X 0,Y 213.225,Z 696.613,A -85,B 0,C 180,E1 7401.807,E2 7401.807} C_VEL
LIN {X 0,Y 221.836,Z 678.694,A -85,B 0,C 180,E1 7400.307,E2 7400.307} C_VEL
LIN {X 0,Y 229.62,Z 659.128,A -85,B 0,C 180,E1 7399.112,E2 7399.112} C_VEL
LIN {X 0,Y 235.854,Z 639.101,A -85,B 0,C 180,E1 7398.2,E2 7398.2} C_VEL
LIN {X 0,Y 240.515,Z 618.355,A -85,B 0,C 180,E1 7397.488,E2 7397.488} C_VEL
LIN {X 0,Y 243.51,Z 596.855,A -85,B 0,C 180,E1 7396.942,E2 7396.942} C_VEL
LIN {X 0,Y 253.906,Z 494.611,A -85,B 0,C 180,E1 7394.772,E2 7394.772} C_VEL
LIN {X 0,Y 250.65,Z 486.073,A -85,B 0,C 180,E1 7391.388,E2 7391.388} C_VEL
LIN {X 0,Y 247.772,Z 479.008,A -85,B 0,C 180,E1 7387.536,E2 7387.536} C_VEL
LIN {X 0,Y 245.813,Z 474.192,A -85,B 0,C 180,E1 7383.731,E2 7383.731} C_VEL
LIN {X 0,Y 244.707,Z 471.127,A -85,B 0,C 180,E1 7379.765,E2 7379.765} C_VEL
LIN {X 0,Y 244.572,Z 470.551,A -85,B 0,C 180,E1 7374.839,E2 7374.839} C_VEL
LIN {X 0,Y 245.601,Z 471.552,A -85,B 0,C 180,E1 7370.864,E2 7370.864} C_VEL
LIN {X 0,Y 247.777,Z 475.718,A -85,B 0,C 180,E1 7366.464,E2 7366.464} C_VEL
LIN {X 0,Y 249.935,Z 479.958,A -85,B 0,C 180,E1 7363.498,E2 7363.498} C_VEL
LIN {X 0,Y 253.156,Z 486.57,A -85,B 0,C 180,E1 7360.07,E2 7360.07} C_VEL
LIN {X 0,Y 254.035,Z 488.817,A -85,B 0,C 180,E1 7359.22,E2 7359.22} C_VEL
LIN {X 0,Y 245.027,Z 582.268,A -85,B 0,C 180,E1 7357.248,E2 7357.248} C_VEL
LIN {X 0,Y 242.417,Z 601.854,A -85,B 0,C 180,E1 7356.59,E2 7356.59} C_VEL
LIN {X 0,Y 238.437,Z 620.741,A -85,B 0,C 180,E1 7355.704,E2 7355.704} C_VEL
LIN {X 0,Y 233.082,Z 639.179,A -85,B 0,C 180,E1 7354.55,E2 7354.55} C_VEL
LIN {X 0,Y 226.079,Z 657.877,A -85,B 0,C 180,E1 7353.016,E2 7353.016} C_VEL
LIN {X 0,Y 217.997,Z 675.305,A -85,B 0,C 180,E1 7351.165,E2 7351.165} C_VEL
LIN {X 0,Y 208.969,Z 691.58,A -85,B 0,C 180,E1 7348.919,E2 7348.919} C_VEL
LIN {X 0,Y 199.111,Z 706.721,A -85,B 0,C 180,E1 7346.207,E2 7346.207} C_VEL
LIN {X 0,Y 188.972,Z 720.256,A -85,B 0,C 180,E1 7343.027,E2 7343.027} C_VEL
LIN {X 0,Y 178.413,Z 732.669,A -85,B 0,C 180,E1 7339.16,E2 7339.16} C_VEL
LIN {X 0,Y 168.042,Z 743.531,A -85,B 0,C 180,E1 7334.595,E2 7334.595} C_VEL
LIN {X 0,Y 158.215,Z 752.852,A -85,B 0,C 180,E1 7329.194,E2 7329.194} C_VEL
LIN {X 0,Y 149.331,Z 760.614,A -85,B 0,C 180,E1 7322.842,E2 7322.842} C_VEL
LIN {X 0,Y 141.877,Z 766.753,A -85,B 0,C 180,E1 7315.46,E2 7315.46} C_VEL
LIN {X 0,Y 136.579,Z 770.991,A -85,B 0,C 180,E1 7307.466,E2 7307.466} C_VEL
LIN {X 0,Y 133.342,Z 773.581,A -85,B 0,C 180,E1 7298.625,E2 7298.625} C_VEL
LIN {X 0,Y 132.383,Z 774.387,A -85,B 0,C 180,E1 7290,E2 7290} C_VEL
LIN {X 0,Y 133.325,Z 773.612,A -85,B 0,C 180,E1 7281.374,E2 7281.374} C_VEL
LIN {X 0,Y 136.332,Z 771.219,A -85,B 0,C 180,E1 7272.941,E2 7272.941} C_VEL
LIN {X 0,Y 141.504,Z 767.104,A -85,B 0,C 180,E1 7264.916,E2 7264.916} C_VEL
LIN {X 0,Y 148.841,Z 761.12,A -85,B 0,C 180,E1 7257.494,E2 7257.494} C_VEL
LIN {X 0,Y 157.628,Z 753.514,A -85,B 0,C 180,E1 7251.101,E2 7251.101} C_VEL
LIN {X 0,Y 167.373,Z 744.349,A -85,B 0,C 180,E1 7245.66,E2 7245.66} C_VEL
LIN {X 0,Y 177.682,Z 733.655,A -85,B 0,C 180,E1 7241.06,E2 7241.06} C_VEL
LIN {X 0,Y 188.193,Z 721.441,A -85,B 0,C 180,E1 7237.163,E2 7237.163} C_VEL
LIN {X 0,Y 197.936,Z 708.614,A -85,B 0,C 180,E1 7234.064,E2 7234.064} C_VEL
LIN {X 0,Y 207.38,Z 694.44,A -85,B 0,C 180,E1 7231.421,E2 7231.421} C_VEL
LIN {X 0,Y 216.376,Z 678.763,A -85,B 0,C 180,E1 7229.152,E2 7229.152} C_VEL
LIN {X 0,Y 224.431,Z 662.127,A -85,B 0,C 180,E1 7227.282,E2 7227.282} C_VEL
LIN {X 0,Y 231.427,Z 644.54,A -85,B 0,C 180,E1 7225.739,E2 7225.739} C_VEL
LIN {X 0,Y 237.288,Z 625.857,A -85,B 0,C 180,E1 7224.477,E2 7224.477} C_VEL
LIN {X 0,Y 241.784,Z 606.454,A -85,B 0,C 180,E1 7223.492,E2 7223.492} C_VEL
LIN {X 0,Y 244.786,Z 586.673,A -85,B 0,C 180,E1 7222.769,E2 7222.769} C_VEL
LIN {X 0,Y 250.009,Z 532.343,A -85,B 0,C 180,E1 7221.543,E2 7221.543} C_VEL
LIN {X 0,Y 254.254,Z 488.678,A -85,B 0,C 180,E1 7220.65,E2 7220.65} C_VEL
LIN {X 0,Y 250.937,Z 481.573,A -85,B 0,C 180,E1 7217.269,E2 7217.269} C_VEL
LIN {X 0,Y 248.614,Z 477.126,A -85,B 0,C 180,E1 7214.32,E2 7214.32} C_VEL
LIN {X 0,Y 247.259,Z 474.553,A -85,B 0,C 180,E1 7212.139,E2 7212.139} C_VEL
LIN {X 0,Y 245.584,Z 471.298,A -85,B 0,C 180,E1 7208.193,E2 7208.193} C_VEL
LIN {X 0,Y 244.724,Z 470.833,A -85,B 0,C 180,E1 7202.811,E2 7202.811} C_VEL
LIN {X 0,Y 245.064,Z 471.614,A -85,B 0,C 180,E1 7199.767,E2 7199.767} C_VEL
LIN {X 0,Y 246.412,Z 475.312,A -85,B 0,C 180,E1 7195.462,E2 7195.462} C_VEL
LIN {X 0,Y 248.546,Z 480.442,A -85,B 0,C 180,E1 7191.674,E2 7191.674} C_VEL
LIN {X 0,Y 251.166,Z 487.048,A -85,B 0,C 180,E1 7188.287,E2 7188.287} C_VEL
LIN {X 0,Y 254.131,Z 494.822,A -85,B 0,C 180,E1 7185.227,E2 7185.227} C_VEL
LIN {X 0,Y 242.245,Z 609.222,A -85,B 0,C 180,E1 7182.786,E2 7182.786} C_VEL
LIN {X 0,Y 238.249,Z 630.425,A -85,B 0,C 180,E1 7182.145,E2 7182.145} C_VEL
LIN {X 0,Y 234.022,Z 646.228,A -85,B 0,C 180,E1 7181.524,E2 7181.524} C_VEL
LIN {X 0,Y 231.339,Z 653.581,A -85,B 0,C 180,E1 7181.417,E2 7181.417} C_VEL
LIN {X 0,Y 222.223,Z 671.527,A -85,B 0,C 180,E1 7181.838,E2 7181.838} C_VEL
LIN {X 0,Y 218.865,Z 678.321,A -85,B 0,C 180,E1 7181.637,E2 7181.637} C_VEL
LIN {X 0,Y 209.474,Z 697.227,A -85,B 0,C 180,E1 7180.1,E2 7180.1} C_VEL
LIN {X 0,Y 199.274,Z 714.635,A -85,B 0,C 180,E1 7178.157,E2 7178.157} C_VEL
LIN {X 0,Y 188.2,Z 731.072,A -85,B 0,C 180,E1 7175.659,E2 7175.659} C_VEL
LIN {X 0,Y 176.835,Z 745.991,A -85,B 0,C 180,E1 7172.583,E2 7172.583} C_VEL
LIN {X 0,Y 165.767,Z 759.117,A -85,B 0,C 180,E1 7168.923,E2 7168.923} C_VEL
LIN {X 0,Y 154.275,Z 771.737,A -85,B 0,C 180,E1 7164.106,E2 7164.106} C_VEL
LIN {X 0,Y 143.565,Z 782.883,A -85,B 0,C 180,E1 7158.174,E2 7158.174} C_VEL
LIN {X 0,Y 134.267,Z 792.519,A -85,B 0,C 180,E1 7150.942,E2 7150.942} C_VEL
LIN {X 0,Y 127.095,Z 800.561,A -85,B 0,C 180,E1 7142.34,E2 7142.34} C_VEL
LIN {X 0,Y 122.95,Z 806.617,A -85,B 0,C 180,E1 7132.975,E2 7132.975} C_VEL
LIN {X 0,Y 121.864,Z 810.769,A -85,B 0,C 180,E1 7123.281,E2 7123.281} C_VEL
LIN {X 0,Y 122.895,Z 812.832,A -85,B 0,C 180,E1 7115.134,E2 7115.134} C_VEL
LIN {X 0,Y 123.784,Z 813.301,A -85,B 0,C 180,E1 7110,E2 7110} C_VEL
LIN {X 0,Y 122.896,Z 812.82,A -85,B 0,C 180,E1 7104.866,E2 7104.866} C_VEL
LIN {X 0,Y 121.864,Z 810.745,A -85,B 0,C 180,E1 7096.719,E2 7096.719} C_VEL
LIN {X 0,Y 122.954,Z 806.574,A -85,B 0,C 180,E1 7087.025,E2 7087.025} C_VEL
LIN {X 0,Y 127.094,Z 800.499,A -85,B 0,C 180,E1 7077.66,E2 7077.66} C_VEL
LIN {X 0,Y 134.264,Z 792.434,A -85,B 0,C 180,E1 7069.057,E2 7069.057} C_VEL
LIN {X 0,Y 143.56,Z 782.769,A -85,B 0,C 180,E1 7061.823,E2 7061.823} C_VEL
LIN {X 0,Y 154.269,Z 771.592,A -85,B 0,C 180,E1 7055.891,E2 7055.891} C_VEL
LIN {X 0,Y 165.761,Z 758.938,A -85,B 0,C 180,E1 7051.073,E2 7051.073} C_VEL
LIN {X 0,Y 177.211,Z 745.277,A -85,B 0,C 180,E1 7047.295,E2 7047.295} C_VEL
LIN {X 0,Y 188.593,Z 730.225,A -85,B 0,C 180,E1 7044.236,E2 7044.236} C_VEL
LIN {X 0,Y 199.265,Z 714.311,A -85,B 0,C 180,E1 7041.836,E2 7041.836} C_VEL
LIN {X 0,Y 209.465,Z 696.83,A -85,B 0,C 180,E1 7039.893,E2 7039.893} C_VEL
LIN {X 0,Y 218.586,Z 678.45,A -85,B 0,C 180,E1 7038.398,E2 7038.398} C_VEL
LIN {X 0,Y 226.645,Z 658.732,A -85,B 0,C 180,E1 7037.239,E2 7037.239} C_VEL
LIN {X 0,Y 233.138,Z 638.339,A -85,B 0,C 180,E1 7036.348,E2 7036.348} C_VEL
LIN {X 0,Y 237.892,Z 617.644,A -85,B 0,C 180,E1 7035.666,E2 7035.666} C_VEL
LIN {X 0,Y 240.959,Z 596.18,A -85,B 0,C 180,E1 7035.137,E2 7035.137} C_VEL
LIN {X 0,Y 251.058,Z 499.141,A -85,B 0,C 180,E1 7033.12,E2 7033.12} C_VEL
LIN {X 0,Y 248.131,Z 491.094,A -85,B 0,C 180,E1 7029.626,E2 7029.626} C_VEL
LIN {X 0,Y 245.995,Z 485.503,A -85,B 0,C 180,E1 7026.3,E2 7026.3} C_VEL
LIN {X 0,Y 244.629,Z 481.893,A -85,B 0,C 180,E1 7023.28,E2 7023.28} C_VEL
LIN {X 0,Y 243.681,Z 479.016,A -85,B 0,C 180,E1 7019.529,E2 7019.529} C_VEL
LIN {X 0,Y 243.628,Z 478.519,A -85,B 0,C 180,E1 7014.583,E2 7014.583} C_VEL
LIN {X 0,Y 244.54,Z 479.475,A -85,B 0,C 180,E1 7011.061,E2 7011.061} C_VEL
LIN {X 0,Y 246.505,Z 483.434,A -85,B 0,C 180,E1 7006.871,E2 7006.871} C_VEL
LIN {X 0,Y 248.58,Z 487.711,A -85,B 0,C 180,E1 7003.886,E2 7003.886} C_VEL
LIN {X 0,Y 251.249,Z 493.513,A -85,B 0,C 180,E1 7000.869,E2 7000.869} C_VEL
LIN {X 0,Y 242.355,Z 583.135,A -85,B 0,C 180,E1 6999.011,E2 6999.011} C_VEL
LIN {X 0,Y 239.66,Z 602.702,A -85,B 0,C 180,E1 6998.364,E2 6998.364} C_VEL
LIN {X 0,Y 235.43,Z 622.086,A -85,B 0,C 180,E1 6997.471,E2 6997.471} C_VEL
LIN {X 0,Y 229.813,Z 640.766,A -85,B 0,C 180,E1 6996.32,E2 6996.32} C_VEL
LIN {X 0,Y 222.797,Z 658.922,A -85,B 0,C 180,E1 6994.859,E2 6994.859} C_VEL
LIN {X 0,Y 214.306,Z 676.668,A -85,B 0,C 180,E1 6993.011,E2 6993.011} C_VEL
LIN {X 0,Y 204.999,Z 692.902,A -85,B 0,C 180,E1 6990.807,E2 6990.807} C_VEL
LIN {X 0,Y 194.828,Z 707.997,A -85,B 0,C 180,E1 6988.138,E2 6988.138} C_VEL
LIN {X 0,Y 184.325,Z 721.512,A -85,B 0,C 180,E1 6984.992,E2 6984.992} C_VEL
LIN {X 0,Y 173.339,Z 733.908,A -85,B 0,C 180,E1 6981.14,E2 6981.14} C_VEL
LIN {X 0,Y 162.495,Z 744.757,A -85,B 0,C 180,E1 6976.557,E2 6976.557} C_VEL
LIN {X 0,Y 152.151,Z 754.071,A -85,B 0,C 180,E1 6971.081,E2 6971.081} C_VEL
LIN {X 0,Y 142.731,Z 761.826,A -85,B 0,C 180,E1 6964.569,E2 6964.569} C_VEL
LIN {X 0,Y 134.757,Z 767.961,A -85,B 0,C 180,E1 6956.91,E2 6956.91} C_VEL
LIN {X 0,Y 129.039,Z 772.197,A -85,B 0,C 180,E1 6948.523,E2 6948.523} C_VEL
LIN {X 0,Y 125.521,Z 774.784,A -85,B 0,C 180,E1 6939.167,E2 6939.167} C_VEL
LIN {X 0,Y 124.474,Z 775.588,A -85,B 0,C 180,E1 6930,E2 6930} C_VEL
LIN {X 0,Y 125.504,Z 774.814,A -85,B 0,C 180,E1 6920.832,E2 6920.832} C_VEL
LIN {X 0,Y 128.775,Z 772.422,A -85,B 0,C 180,E1 6911.907,E2 6911.907} C_VEL
LIN {X 0,Y 134.36,Z 768.308,A -85,B 0,C 180,E1 6903.482,E2 6903.482} C_VEL
LIN {X 0,Y 141.767,Z 762.656,A -85,B 0,C 180,E1 6896.141,E2 6896.141} C_VEL
LIN {X 0,Y 151.002,Z 755.155,A -85,B 0,C 180,E1 6889.542,E2 6889.542} C_VEL
LIN {X 0,Y 161.192,Z 746.108,A -85,B 0,C 180,E1 6883.986,E2 6883.986} C_VEL
LIN {X 0,Y 171.921,Z 735.549,A -85,B 0,C 180,E1 6879.333,E2 6879.333} C_VEL
LIN {X 0,Y 182.816,Z 723.493,A -85,B 0,C 180,E1 6875.424,E2 6875.424} C_VEL
LIN {X 0,Y 193.535,Z 709.99,A -85,B 0,C 180,E1 6872.15,E2 6872.15} C_VEL
LIN {X 0,Y 203.376,Z 695.74,A -85,B 0,C 180,E1 6869.523,E2 6869.523} C_VEL
LIN {X 0,Y 212.646,Z 680.114,A -85,B 0,C 180,E1 6867.296,E2 6867.296} C_VEL
LIN {X 0,Y 221.33,Z 662.676,A -85,B 0,C 180,E1 6865.382,E2 6865.382} C_VEL
LIN {X 0,Y 228.522,Z 644.98,A -85,B 0,C 180,E1 6863.877,E2 6863.877} C_VEL
LIN {X 0,Y 234.545,Z 626.145,A -85,B 0,C 180,E1 6862.645,E2 6862.645} C_VEL
LIN {X 0,Y 239.215,Z 606.245,A -85,B 0,C 180,E1 6861.672,E2 6861.672} C_VEL
LIN {X 0,Y 242.276,Z 586.007,A -85,B 0,C 180,E1 6860.962,E2 6860.962} C_VEL
LIN {X 0,Y 248.182,Z 526.446,A -85,B 0,C 180,E1 6859.669,E2 6859.669} C_VEL
LIN {X 0,Y 251.427,Z 493.586,A -85,B 0,C 180,E1 6858.972,E2 6858.972} C_VEL
LIN {X 0,Y 248.549,Z 487.313,A -85,B 0,C 180,E1 6855.637,E2 6855.637} C_VEL
LIN {X 0,Y 246.304,Z 482.635,A -85,B 0,C 180,E1 6852.187,E2 6852.187} C_VEL
LIN {X 0,Y 244.548,Z 479.2,A -85,B 0,C 180,E1 6847.991,E2 6847.991} C_VEL
LIN {X 0,Y 243.742,Z 478.774,A -85,B 0,C 180,E1 6842.822,E2 6842.822} C_VEL
LIN {X 0,Y 244.03,Z 479.5,A -85,B 0,C 180,E1 6840,E2 6840} C_VEL
LIN {X 0,Y 245.205,Z 482.992,A -85,B 0,C 180,E1 6835.908,E2 6835.908} C_VEL
LIN {X 0,Y 247.12,Z 487.976,A -85,B 0,C 180,E1 6832.211,E2 6832.211} C_VEL
LIN {X 0,Y 249.46,Z 494.293,A -85,B 0,C 180,E1 6828.967,E2 6828.967} C_VEL
LIN {X 0,Y 251.264,Z 499.644,A -85,B 0,C 180,E1 6826.863,E2 6826.863} C_VEL
LIN {X 0,Y 239.688,Z 608.346,A -85,B 0,C 180,E1 6824.603,E2 6824.603} C_VEL
LIN {X 0,Y 235.654,Z 629.381,A -85,B 0,C 180,E1 6823.991,E2 6823.991} C_VEL
LIN {X 0,Y 230.013,Z 649.616,A -85,B 0,C 180,E1 6823.214,E2 6823.214} C_VEL
LIN {X 0,Y 222.632,Z 669.643,A -85,B 0,C 180,E1 6822.191,E2 6822.191} C_VEL
LIN {X 0,Y 218.865,Z 678.321,A -85,B 0,C 180,E1 6821.637,E2 6821.637} C_VEL
LIN {X 0,Y 215.317,Z 685.172,A -85,B 0,C 180,E1 6821.39,E2 6821.39} C_VEL
LIN {X 0,Y 204.558,Z 700.844,A -85,B 0,C 180,E1 6821.432,E2 6821.432} C_VEL
LIN {X 0,Y 200.213,Z 707.158,A -85,B 0,C 180,E1 6821.081,E2 6821.081} C_VEL
LIN {X 0,Y 199.642,Z 708.04,A -85,B 0,C 180,E1 6820.987,E2 6820.987} C_VEL
LIN {X 0,Y 189.376,Z 723.627,A -85,B 0,C 180,E1 6818.96,E2 6818.96} C_VEL
LIN {X 0,Y 177.583,Z 739.321,A -85,B 0,C 180,E1 6816.193,E2 6816.193} C_VEL
LIN {X 0,Y 165.116,Z 754.037,A -85,B 0,C 180,E1 6812.6,E2 6812.6} C_VEL
LIN {X 0,Y 152.981,Z 767.021,A -85,B 0,C 180,E1 6808.171,E2 6808.171} C_VEL
LIN {X 0,Y 141.012,Z 778.903,A -85,B 0,C 180,E1 6802.427,E2 6802.427} C_VEL
LIN {X 0,Y 130.5,Z 788.962,A -85,B 0,C 180,E1 6795.44,E2 6795.44} C_VEL
LIN {X 0,Y 121.838,Z 797.526,A -85,B 0,C 180,E1 6786.802,E2 6786.802} C_VEL
LIN {X 0,Y 116.251,Z 804.077,A -85,B 0,C 180,E1 6777.118,E2 6777.118} C_VEL
LIN {X 0,Y 113.97,Z 808.695,A -85,B 0,C 180,E1 6766.828,E2 6766.828} C_VEL
LIN {X 0,Y 114.5,Z 811.206,A -85,B 0,C 180,E1 6757.526,E2 6757.526} C_VEL
LIN {X 0,Y 115.769,Z 812.044,A -85,B 0,C 180,E1 6750.99,E2 6750.99} C_VEL
LIN {X 0,Y 115.497,Z 811.914,A -85,B 0,C 180,E1 6747.519,E2 6747.519} C_VEL
LIN {X 0,Y 114.081,Z 810.561,A -85,B 0,C 180,E1 6739.394,E2 6739.394} C_VEL
LIN {X 0,Y 114.391,Z 807.231,A -85,B 0,C 180,E1 6729.536,E2 6729.536} C_VEL
LIN {X 0,Y 117.589,Z 802.212,A -85,B 0,C 180,E1 6719.89,E2 6719.89} C_VEL
LIN {X 0,Y 124.135,Z 795.049,A -85,B 0,C 180,E1 6710.484,E2 6710.484} C_VEL
LIN {X 0,Y 133.222,Z 786.193,A -85,B 0,C 180,E1 6702.489,E2 6702.489} C_VEL
LIN {X 0,Y 144.278,Z 775.535,A -85,B 0,C 180,E1 6695.826,E2 6695.826} C_VEL
LIN {X 0,Y 155.791,Z 763.869,A -85,B 0,C 180,E1 6690.686,E2 6690.686} C_VEL
LIN {X 0,Y 167.847,Z 750.69,A -85,B 0,C 180,E1 6686.536,E2 6686.536} C_VEL
LIN {X 0,Y 179.659,Z 736.401,A -85,B 0,C 180,E1 6683.274,E2 6683.274} C_VEL
LIN {X 0,Y 190.819,Z 721.24,A -85,B 0,C 180,E1 6680.726,E2 6680.726} C_VEL
LIN {X 0,Y 201.564,Z 704.565,A -85,B 0,C 180,E1 6678.661,E2 6678.661} C_VEL
LIN {X 0,Y 211.361,Z 686.846,A -85,B 0,C 180,E1 6677.055,E2 6677.055} C_VEL
LIN {X 0,Y 220.062,Z 668.056,A -85,B 0,C 180,E1 6675.819,E2 6675.819} C_VEL
LIN {X 0,Y 227.565,Z 647.862,A -85,B 0,C 180,E1 6674.852,E2 6674.852} C_VEL
LIN {X 0,Y 233.312,Z 627.289,A -85,B 0,C 180,E1 6674.109,E2 6674.109} C_VEL
LIN {X 0,Y 237.313,Z 606.212,A -85,B 0,C 180,E1 6673.531,E2 6673.531} C_VEL
LIN {X 0,Y 248.415,Z 503.894,A -85,B 0,C 180,E1 6671.452,E2 6671.452} C_VEL
LIN {X 0,Y 246.22,Z 497.525,A -85,B 0,C 180,E1 6668.465,E2 6668.465} C_VEL
LIN {X 0,Y 244.596,Z 492.903,A -85,B 0,C 180,E1 6665.63,E2 6665.63} C_VEL
LIN {X 0,Y 243.455,Z 489.593,A -85,B 0,C 180,E1 6662.824,E2 6662.824} C_VEL
LIN {X 0,Y 242.665,Z 486.908,A -85,B 0,C 180,E1 6659.291,E2 6659.291} C_VEL
LIN {X 0,Y 242.657,Z 486.463,A -85,B 0,C 180,E1 6654.561,E2 6654.561} C_VEL
LIN {X 0,Y 243.447,Z 487.289,A -85,B 0,C 180,E1 6651.378,E2 6651.378} C_VEL
LIN {X 0,Y 245.246,Z 491.15,A -85,B 0,C 180,E1 6647.281,E2 6647.281} C_VEL
LIN {X 0,Y 247.287,Z 495.563,A -85,B 0,C 180,E1 6644.213,E2 6644.213} C_VEL
LIN {X 0,Y 248.611,Z 498.871,A -85,B 0,C 180,E1 6642.538,E2 6642.538} C_VEL
LIN {X 0,Y 239.939,Z 583.793,A -85,B 0,C 180,E1 6640.816,E2 6640.816} C_VEL
LIN {X 0,Y 237.164,Z 603.419,A -85,B 0,C 180,E1 6640.183,E2 6640.183} C_VEL
LIN {X 0,Y 232.949,Z 622.393,A -85,B 0,C 180,E1 6639.337,E2 6639.337} C_VEL
LIN {X 0,Y 227.183,Z 641.204,A -85,B 0,C 180,E1 6638.219,E2 6638.219} C_VEL
LIN {X 0,Y 219.793,Z 659.877,A -85,B 0,C 180,E1 6636.764,E2 6636.764} C_VEL
LIN {X 0,Y 211.251,Z 677.308,A -85,B 0,C 180,E1 6635.006,E2 6635.006} C_VEL
LIN {X 0,Y 201.648,Z 693.632,A -85,B 0,C 180,E1 6632.859,E2 6632.859} C_VEL
LIN {X 0,Y 191.16,Z 708.768,A -85,B 0,C 180,E1 6630.254,E2 6630.254} C_VEL
LIN {X 0,Y 179.903,Z 722.764,A -85,B 0,C 180,E1 6627.055,E2 6627.055} C_VEL
LIN {X 0,Y 168.485,Z 735.143,A -85,B 0,C 180,E1 6623.237,E2 6623.237} C_VEL
LIN {X 0,Y 157.151,Z 745.983,A -85,B 0,C 180,E1 6618.655,E2 6618.655} C_VEL
LIN {X 0,Y 146.265,Z 755.289,A -85,B 0,C 180,E1 6613.124,E2 6613.124} C_VEL
LIN {X 0,Y 136.273,Z 763.038,A -85,B 0,C 180,E1 6606.462,E2 6606.462} C_VEL
LIN {X 0,Y 127.733,Z 769.169,A -85,B 0,C 180,E1 6598.521,E2 6598.521} C_VEL
LIN {X 0,Y 121.549,Z 773.402,A -85,B 0,C 180,E1 6589.71,E2 6589.71} C_VEL
LIN {X 0,Y 117.713,Z 775.986,A -85,B 0,C 180,E1 6579.781,E2 6579.781} C_VEL
LIN {X 0,Y 116.565,Z 776.79,A -85,B 0,C 180,E1 6570,E2 6570} C_VEL
LIN {X 0,Y 117.695,Z 776.016,A -85,B 0,C 180,E1 6560.218,E2 6560.218} C_VEL
LIN {X 0,Y 121.265,Z 773.625,A -85,B 0,C 180,E1 6550.743,E2 6550.743} C_VEL
LIN {X 0,Y 127.31,Z 769.512,A -85,B 0,C 180,E1 6541.887,E2 6541.887} C_VEL
LIN {X 0,Y 135.25,Z 763.862,A -85,B 0,C 180,E1 6534.267,E2 6534.267} C_VEL
LIN {X 0,Y 145.057,Z 756.365,A -85,B 0,C 180,E1 6527.509,E2 6527.509} C_VEL
LIN {X 0,Y 155.792,Z 747.325,A -85,B 0,C 180,E1 6521.888,E2 6521.888} C_VEL
LIN {X 0,Y 167.014,Z 736.776,A -85,B 0,C 180,E1 6517.231,E2 6517.231} C_VEL
LIN {X 0,Y 178.346,Z 724.735,A -85,B 0,C 180,E1 6513.352,E2 6513.352} C_VEL
LIN {X 0,Y 188.773,Z 712.122,A -85,B 0,C 180,E1 6510.308,E2 6510.308} C_VEL
LIN {X 0,Y 199.605,Z 697.039,A -85,B 0,C 180,E1 6507.551,E2 6507.551} C_VEL
LIN {X 0,Y 209.36,Z 681.087,A -85,B 0,C 180,E1 6505.33,E2 6505.33} C_VEL
LIN {X 0,Y 218.091,Z 664.058,A -85,B 0,C 180,E1 6503.508,E2 6503.508} C_VEL
LIN {X 0,Y 225.453,Z 646.525,A -85,B 0,C 180,E1 6502.049,E2 6502.049} C_VEL
LIN {X 0,Y 231.634,Z 627.886,A -85,B 0,C 180,E1 6500.852,E2 6500.852} C_VEL
LIN {X 0,Y 236.407,Z 608.474,A -85,B 0,C 180,E1 6499.912,E2 6499.912} C_VEL
LIN {X 0,Y 239.62,Z 588.738,A -85,B 0,C 180,E1 6499.214,E2 6499.214} C_VEL
LIN {X 0,Y 244.839,Z 537.832,A -85,B 0,C 180,E1 6498.097,E2 6498.097} C_VEL
LIN {X 0,Y 248.836,Z 498.724,A -85,B 0,C 180,E1 6497.299,E2 6497.299} C_VEL
LIN {X 0,Y 246.359,Z 493.117,A -85,B 0,C 180,E1 6493.975,E2 6493.975} C_VEL
LIN {X 0,Y 244.838,Z 489.99,A -85,B 0,C 180,E1 6491.305,E2 6491.305} C_VEL
LIN {X 0,Y 243.503,Z 487.102,A -85,B 0,C 180,E1 6487.788,E2 6487.788} C_VEL
LIN {X 0,Y 242.773,Z 486.747,A -85,B 0,C 180,E1 6482.597,E2 6482.597} C_VEL
LIN {X 0,Y 243.007,Z 487.386,A -85,B 0,C 180,E1 6480.236,E2 6480.236} C_VEL
LIN {X 0,Y 244.049,Z 490.824,A -85,B 0,C 180,E1 6476.242,E2 6476.242} C_VEL
LIN {X 0,Y 245.714,Z 495.533,A -85,B 0,C 180,E1 6472.754,E2 6472.754} C_VEL
LIN {X 0,Y 247.827,Z 501.665,A -85,B 0,C 180,E1 6469.599,E2 6469.599} C_VEL
LIN {X 0,Y 248.637,Z 504.328,A -85,B 0,C 180,E1 6468.54,E2 6468.54} C_VEL
LIN {X 0,Y 237.373,Z 607.494,A -85,B 0,C 180,E1 6466.457,E2 6466.457} C_VEL
LIN {X 0,Y 233.244,Z 628.586,A -85,B 0,C 180,E1 6465.869,E2 6465.869} C_VEL
LIN {X 0,Y 227.574,Z 648.582,A -85,B 0,C 180,E1 6465.139,E2 6465.139} C_VEL
LIN {X 0,Y 220.187,Z 668.326,A -85,B 0,C 180,E1 6464.19,E2 6464.19} C_VEL
LIN {X 0,Y 211.279,Z 687.467,A -85,B 0,C 180,E1 6462.924,E2 6462.924} C_VEL
LIN {X 0,Y 201.137,Z 705.669,A -85,B 0,C 180,E1 6461.254,E2 6461.254} C_VEL
LIN {X 0,Y 199.642,Z 708.04,A -85,B 0,C 180,E1 6460.987,E2 6460.987} C_VEL
LIN {X 0,Y 195.24,Z 714.33,A -85,B 0,C 180,E1 6460.507,E2 6460.507} C_VEL
LIN {X 0,Y 181.875,Z 729.241,A -85,B 0,C 180,E1 6459.977,E2 6459.977} C_VEL
LIN {X 0,Y 177.003,Z 734.779,A -85,B 0,C 180,E1 6459.281,E2 6459.281} C_VEL
LIN {X 0,Y 164.973,Z 748.868,A -85,B 0,C 180,E1 6456.226,E2 6456.226} C_VEL
LIN {X 0,Y 152.301,Z 762.168,A -85,B 0,C 180,E1 6452.218,E2 6452.218} C_VEL
LIN {X 0,Y 139.57,Z 774.389,A -85,B 0,C 180,E1 6446.945,E2 6446.945} C_VEL
LIN {X 0,Y 127.589,Z 785.152,A -85,B 0,C 180,E1 6440.171,E2 6440.171} C_VEL
LIN {X 0,Y 117.375,Z 794.256,A -85,B 0,C 180,E1 6431.638,E2 6431.638} C_VEL
LIN {X 0,Y 110.187,Z 801.303,A -85,B 0,C 180,E1 6421.755,E2 6421.755} C_VEL
LIN {X 0,Y 106.474,Z 806.421,A -85,B 0,C 180,E1 6410.906,E2 6410.906} C_VEL
LIN {X 0,Y 106.167,Z 809.553,A -85,B 0,C 180,E1 6400.307,E2 6400.307} C_VEL
LIN {X 0,Y 107.607,Z 810.749,A -85,B 0,C 180,E1 6392.13,E2 6392.13} C_VEL
LIN {X 0,Y 107.895,Z 810.868,A -85,B 0,C 180,E1 6389.469,E2 6389.469} C_VEL
LIN {X 0,Y 106.454,Z 809.957,A -85,B 0,C 180,E1 6381.901,E2 6381.901} C_VEL
LIN {X 0,Y 106.107,Z 807.406,A -85,B 0,C 180,E1 6371.883,E2 6371.883} C_VEL
LIN {X 0,Y 108.924,Z 802.762,A -85,B 0,C 180,E1 6360.889,E2 6360.889} C_VEL
LIN {X 0,Y 115.268,Z 796.19,A -85,B 0,C 180,E1 6350.713,E2 6350.713} C_VEL
LIN {X 0,Y 124.779,Z 787.589,A -85,B 0,C 180,E1 6341.825,E2 6341.825} C_VEL
LIN {X 0,Y 136.227,Z 777.367,A -85,B 0,C 180,E1 6334.713,E2 6334.713} C_VEL
LIN {X 0,Y 148.753,Z 765.575,A -85,B 0,C 180,E1 6329.099,E2 6329.099} C_VEL
LIN {X 0,Y 161.767,Z 752.23,A -85,B 0,C 180,E1 6324.693,E2 6324.693} C_VEL
LIN {X 0,Y 174.408,Z 737.778,A -85,B 0,C 180,E1 6321.32,E2 6321.32} C_VEL
LIN {X 0,Y 186.765,Z 721.753,A -85,B 0,C 180,E1 6318.638,E2 6318.638} C_VEL
LIN {X 0,Y 198.205,Z 704.643,A -85,B 0,C 180,E1 6316.576,E2 6316.576} C_VEL
LIN {X 0,Y 208.478,Z 686.612,A -85,B 0,C 180,E1 6315.009,E2 6315.009} C_VEL
LIN {X 0,Y 217.744,Z 667.053,A -85,B 0,C 180,E1 6313.795,E2 6313.795} C_VEL
LIN {X 0,Y 225.4,Z 646.768,A -85,B 0,C 180,E1 6312.886,E2 6312.886} C_VEL
LIN {X 0,Y 231.205,Z 626.288,A -85,B 0,C 180,E1 6312.189,E2 6312.189} C_VEL
LIN {X 0,Y 235.253,Z 605.32,A -85,B 0,C 180,E1 6311.642,E2 6311.642} C_VEL
LIN {X 0,Y 245.951,Z 508.72,A -85,B 0,C 180,E1 6309.712,E2 6309.712} C_VEL
LIN {X 0,Y 244.101,Z 502.858,A -85,B 0,C 180,E1 6306.703,E2 6306.703} C_VEL
LIN {X 0,Y 242.489,Z 497.782,A -85,B 0,C 180,E1 6302.954,E2 6302.954} C_VEL
LIN {X 0,Y 241.653,Z 494.801,A -85,B 0,C 180,E1 6299.051,E2 6299.051} C_VEL
LIN {X 0,Y 241.686,Z 494.409,A -85,B 0,C 180,E1 6294.539,E2 6294.539} C_VEL
LIN {X 0,Y 242.394,Z 495.209,A -85,B 0,C 180,E1 6291.579,E2 6291.579} C_VEL
LIN {X 0,Y 244.01,Z 498.865,A -85,B 0,C 180,E1 6287.697,E2 6287.697} C_VEL
LIN {X 0,Y 246.034,Z 503.479,A -85,B 0,C 180,E1 6284.502,E2 6284.502} C_VEL
LIN {X 0,Y 246.186,Z 504.23,A -85,B 0,C 180,E1 6284.243,E2 6284.243} C_VEL
LIN {X 0,Y 237.734,Z 584.723,A -85,B 0,C 180,E1 6282.649,E2 6282.649} C_VEL
LIN {X 0,Y 234.859,Z 604.39,A -85,B 0,C 180,E1 6282.028,E2 6282.028} C_VEL
LIN {X 0,Y 230.507,Z 623.429,A -85,B 0,C 180,E1 6281.203,E2 6281.203} C_VEL
LIN {X 0,Y 224.806,Z 641.606,A -85,B 0,C 180,E1 6280.161,E2 6280.161} C_VEL
LIN {X 0,Y 217.408,Z 659.997,A -85,B 0,C 180,E1 6278.79,E2 6278.79} C_VEL
LIN {X 0,Y 208.871,Z 677.148,A -85,B 0,C 180,E1 6277.141,E2 6277.141} C_VEL
LIN {X 0,Y 199.409,Z 693.004,A -85,B 0,C 180,E1 6275.166,E2 6275.166} C_VEL
LIN {X 0,Y 188.947,Z 707.92,A -85,B 0,C 180,E1 6272.746,E2 6272.746} C_VEL
LIN {X 0,Y 178.011,Z 721.363,A -85,B 0,C 180,E1 6269.879,E2 6269.879} C_VEL
LIN {X 0,Y 166.769,Z 733.436,A -85,B 0,C 180,E1 6266.444,E2 6266.444} C_VEL
LIN {X 0,Y 154.73,Z 744.788,A -85,B 0,C 180,E1 6262.03,E2 6262.03} C_VEL
LIN {X 0,Y 143.009,Z 754.559,A -85,B 0,C 180,E1 6256.644,E2 6256.644} C_VEL
LIN {X 0,Y 132.064,Z 762.73,A -85,B 0,C 180,E1 6250.055,E2 6250.055} C_VEL
LIN {X 0,Y 122.886,Z 768.976,A -85,B 0,C 180,E1 6242.479,E2 6242.479} C_VEL
LIN {X 0,Y 115.542,Z 773.666,A -85,B 0,C 180,E1 6233.457,E2 6233.457} C_VEL
LIN {X 0,Y 110.806,Z 776.59,A -85,B 0,C 180,E1 6223.568,E2 6223.568} C_VEL
LIN {X 0,Y 108.761,Z 777.868,A -85,B 0,C 180,E1 6213.162,E2 6213.162} C_VEL
LIN {X 0,Y 109.169,Z 777.64,A -85,B 0,C 180,E1 6203.162,E2 6203.162} C_VEL
LIN {X 0,Y 111.919,Z 775.987,A -85,B 0,C 180,E1 6193.389,E2 6193.389} C_VEL
LIN {X 0,Y 117.435,Z 772.592,A -85,B 0,C 180,E1 6183.722,E2 6183.722} C_VEL
LIN {X 0,Y 125.513,Z 767.375,A -85,B 0,C 180,E1 6175.002,E2 6175.002} C_VEL
LIN {X 0,Y 135.283,Z 760.595,A -85,B 0,C 180,E1 6167.736,E2 6167.736} C_VEL
LIN {X 0,Y 146.709,Z 751.805,A -85,B 0,C 180,E1 6161.44,E2 6161.44} C_VEL
LIN {X 0,Y 158.107,Z 742.009,A -85,B 0,C 180,E1 6156.571,E2 6156.571} C_VEL
LIN {X 0,Y 170.379,Z 730.03,A -85,B 0,C 180,E1 6152.325,E2 6152.325} C_VEL
LIN {X 0,Y 181.794,Z 717.27,A -85,B 0,C 180,E1 6149.018,E2 6149.018} C_VEL
LIN {X 0,Y 193.26,Z 702.447,A -85,B 0,C 180,E1 6146.156,E2 6146.156} C_VEL
LIN {X 0,Y 203.835,Z 686.379,A -85,B 0,C 180,E1 6143.823,E2 6143.823} C_VEL
LIN {X 0,Y 212.963,Z 669.874,A -85,B 0,C 180,E1 6141.993,E2 6141.993} C_VEL
LIN {X 0,Y 221.36,Z 651.372,A -85,B 0,C 180,E1 6140.409,E2 6140.409} C_VEL
LIN {X 0,Y 228.074,Z 632.648,A -85,B 0,C 180,E1 6139.181,E2 6139.181} C_VEL
LIN {X 0,Y 233.423,Z 612.684,A -85,B 0,C 180,E1 6138.192,E2 6138.192} C_VEL
LIN {X 0,Y 237.08,Z 592.394,A -85,B 0,C 180,E1 6137.457,E2 6137.457} C_VEL
LIN {X 0,Y 241.701,Z 549.071,A -85,B 0,C 180,E1 6136.479,E2 6136.479} C_VEL
LIN {X 0,Y 246.448,Z 504.107,A -85,B 0,C 180,E1 6135.61,E2 6135.61} C_VEL
LIN {X 0,Y 244.598,Z 499.812,A -85,B 0,C 180,E1 6132.753,E2 6132.753} C_VEL
LIN {X 0,Y 243.524,Z 497.514,A -85,B 0,C 180,E1 6130.648,E2 6130.648} C_VEL
LIN {X 0,Y 242.461,Z 495.005,A -85,B 0,C 180,E1 6127.583,E2 6127.583} C_VEL
LIN {X 0,Y 241.799,Z 494.691,A -85,B 0,C 180,E1 6122.608,E2 6122.608} C_VEL
LIN {X 0,Y 242.015,Z 495.465,A -85,B 0,C 180,E1 6120.237,E2 6120.237} C_VEL
LIN {X 0,Y 242.9,Z 498.654,A -85,B 0,C 180,E1 6116.579,E2 6116.579} C_VEL
LIN {X 0,Y 244.31,Z 502.981,A -85,B 0,C 180,E1 6113.361,E2 6113.361} C_VEL
LIN {X 0,Y 246.184,Z 508.907,A -85,B 0,C 180,E1 6110.297,E2 6110.297} C_VEL
LIN {X 0,Y 235.312,Z 606.641,A -85,B 0,C 180,E1 6108.345,E2 6108.345} C_VEL
LIN {X 0,Y 231.103,Z 627.741,A -85,B 0,C 180,E1 6107.785,E2 6107.785} C_VEL
LIN {X 0,Y 225.335,Z 647.729,A -85,B 0,C 180,E1 6107.097,E2 6107.097} C_VEL
LIN {X 0,Y 217.878,Z 667.319,A -85,B 0,C 180,E1 6106.214,E2 6106.214} C_VEL
LIN {X 0,Y 209.031,Z 686.009,A -85,B 0,C 180,E1 6105.061,E2 6105.061} C_VEL
LIN {X 0,Y 198.657,Z 704.279,A -85,B 0,C 180,E1 6103.491,E2 6103.491} C_VEL
LIN {X 0,Y 187.205,Z 721.443,A -85,B 0,C 180,E1 6101.44,E2 6101.44} C_VEL
LIN {X 0,Y 177.003,Z 734.779,A -85,B 0,C 180,E1 6099.281,E2 6099.281} C_VEL
LIN {X 0,Y 172.013,Z 740.25,A -85,B 0,C 180,E1 6098.5,E2 6098.5} C_VEL
LIN {X 0,Y 157.064,Z 753.161,A -85,B 0,C 180,E1 6097.167,E2 6097.167} C_VEL
LIN {X 0,Y 151.738,Z 757.922,A -85,B 0,C 180,E1 6096.048,E2 6096.048} C_VEL
LIN {X 0,Y 138.112,Z 770.609,A -85,B 0,C 180,E1 6091.157,E2 6091.157} C_VEL
LIN {X 0,Y 125.393,Z 781.479,A -85,B 0,C 180,E1 6084.963,E2 6084.963} C_VEL
LIN {X 0,Y 113.8,Z 790.964,A -85,B 0,C 180,E1 6076.821,E2 6076.821} C_VEL
LIN {X 0,Y 104.747,Z 798.638,A -85,B 0,C 180,E1 6066.698,E2 6066.698} C_VEL
LIN {X 0,Y 99.357,Z 804.341,A -85,B 0,C 180,E1 6055.002,E2 6055.002} C_VEL
LIN {X 0,Y 98.035,Z 807.959,A -85,B 0,C 180,E1 6042.966,E2 6042.966} C_VEL
LIN {X 0,Y 99.472,Z 809.483,A -85,B 0,C 180,E1 6032.881,E2 6032.881} C_VEL
LIN {X 0,Y 99.955,Z 809.662,A -85,B 0,C 180,E1 6029.427,E2 6029.427} C_VEL
LIN {X 0,Y 98.402,Z 808.721,A -85,B 0,C 180,E1 6021.233,E2 6021.233} C_VEL
LIN {X 0,Y 98.378,Z 805.947,A -85,B 0,C 180,E1 6009.785,E2 6009.785} C_VEL
LIN {X 0,Y 101.741,Z 801.496,A -85,B 0,C 180,E1 5998.611,E2 5998.611} C_VEL
LIN {X 0,Y 108.939,Z 794.918,A -85,B 0,C 180,E1 5987.934,E2 5987.934} C_VEL
LIN {X 0,Y 119.373,Z 786.31,A -85,B 0,C 180,E1 5978.836,E2 5978.836} C_VEL
LIN {X 0,Y 131.66,Z 776.083,A -85,B 0,C 180,E1 5971.73,E2 5971.73} C_VEL
LIN {X 0,Y 144.968,Z 764.203,A -85,B 0,C 180,E1 5966.193,E2 5966.193} C_VEL
LIN {X 0,Y 158.486,Z 750.924,A -85,B 0,C 180,E1 5961.972,E2 5961.972} C_VEL
LIN {X 0,Y 171.581,Z 736.457,A -85,B 0,C 180,E1 5958.753,E2 5958.753} C_VEL
LIN {X 0,Y 184.302,Z 720.399,A -85,B 0,C 180,E1 5956.216,E2 5956.216} C_VEL
LIN {X 0,Y 196.026,Z 703.244,A -85,B 0,C 180,E1 5954.282,E2 5954.282} C_VEL
LIN {X 0,Y 206.61,Z 684.97,A -85,B 0,C 180,E1 5952.812,E2 5952.812} C_VEL
LIN {X 0,Y 215.484,Z 666.559,A -85,B 0,C 180,E1 5951.755,E2 5951.755} C_VEL
LIN {X 0,Y 223.249,Z 646.468,A -85,B 0,C 180,E1 5950.911,E2 5950.911} C_VEL
LIN {X 0,Y 229.274,Z 625.681,A -85,B 0,C 180,E1 5950.246,E2 5950.246} C_VEL
LIN {X 0,Y 233.44,Z 604.543,A -85,B 0,C 180,E1 5949.724,E2 5949.724} C_VEL
LIN {X 0,Y 243.717,Z 513.688,A -85,B 0,C 180,E1 5947.958,E2 5947.958} C_VEL
LIN {X 0,Y 242.107,Z 508.248,A -85,B 0,C 180,E1 5944.737,E2 5944.737} C_VEL
LIN {X 0,Y 241.151,Z 504.989,A -85,B 0,C 180,E1 5941.9,E2 5941.9} C_VEL
LIN {X 0,Y 240.632,Z 502.694,A -85,B 0,C 180,E1 5938.809,E2 5938.809} C_VEL
LIN {X 0,Y 240.752,Z 502.382,A -85,B 0,C 180,E1 5934.279,E2 5934.279} C_VEL
LIN {X 0,Y 241.343,Z 503.129,A -85,B 0,C 180,E1 5931.782,E2 5931.782} C_VEL
LIN {X 0,Y 242.787,Z 506.581,A -85,B 0,C 180,E1 5928.117,E2 5928.117} C_VEL
LIN {X 0,Y 243.97,Z 509.678,A -85,B 0,C 180,E1 5925.979,E2 5925.979} C_VEL
LIN {X 0,Y 235.774,Z 585.685,A -85,B 0,C 180,E1 5924.514,E2 5924.514} C_VEL
LIN {X 0,Y 232.802,Z 605.363,A -85,B 0,C 180,E1 5923.908,E2 5923.908} C_VEL
LIN {X 0,Y 228.314,Z 624.463,A -85,B 0,C 180,E1 5923.108,E2 5923.108} C_VEL
LIN {X 0,Y 222.262,Z 643.224,A -85,B 0,C 180,E1 5922.067,E2 5922.067} C_VEL
LIN {X 0,Y 214.501,Z 661.875,A -85,B 0,C 180,E1 5920.716,E2 5920.716} C_VEL
LIN {X 0,Y 205.514,Z 679.31,A -85,B 0,C 180,E1 5919.081,E2 5919.081} C_VEL
LIN {X 0,Y 195.394,Z 695.62,A -85,B 0,C 180,E1 5917.081,E2 5917.081} C_VEL
LIN {X 0,Y 184.049,Z 711.054,A -85,B 0,C 180,E1 5914.584,E2 5914.584} C_VEL
LIN {X 0,Y 171.814,Z 725.261,A -85,B 0,C 180,E1 5911.487,E2 5911.487} C_VEL
LIN {X 0,Y 159.514,Z 737.609,A -85,B 0,C 180,E1 5907.799,E2 5907.799} C_VEL
LIN {X 0,Y 147.058,Z 748.516,A -85,B 0,C 180,E1 5903.249,E2 5903.249} C_VEL
LIN {X 0,Y 134.743,Z 757.997,A -85,B 0,C 180,E1 5897.524,E2 5897.524} C_VEL
LIN {X 0,Y 123.326,Z 765.806,A -85,B 0,C 180,E1 5890.434,E2 5890.434} C_VEL
LIN {X 0,Y 113.613,Z 771.822,A -85,B 0,C 180,E1 5881.872,E2 5881.872} C_VEL
LIN {X 0,Y 106.463,Z 775.965,A -85,B 0,C 180,E1 5872.065,E2 5872.065} C_VEL
LIN {X 0,Y 102.147,Z 778.391,A -85,B 0,C 180,E1 5861.289,E2 5861.289} C_VEL
LIN {X 0,Y 100.746,Z 779.193,A -85,B 0,C 180,E1 5850,E2 5850} C_VEL
LIN {X 0,Y 102.128,Z 778.419,A -85,B 0,C 180,E1 5838.709,E2 5838.709} C_VEL
LIN {X 0,Y 106.426,Z 776.031,A -85,B 0,C 180,E1 5827.927,E2 5827.927} C_VEL
LIN {X 0,Y 113.559,Z 771.921,A -85,B 0,C 180,E1 5818.111,E2 5818.111} C_VEL
LIN {X 0,Y 122.718,Z 766.274,A -85,B 0,C 180,E1 5809.936,E2 5809.936} C_VEL
LIN {X 0,Y 133.787,Z 758.784,A -85,B 0,C 180,E1 5802.914,E2 5802.914} C_VEL
LIN {X 0,Y 145.685,Z 749.755,A -85,B 0,C 180,E1 5797.24,E2 5797.24} C_VEL
LIN {X 0,Y 157.934,Z 739.226,A -85,B 0,C 180,E1 5792.65,E2 5792.65} C_VEL
LIN {X 0,Y 170.16,Z 727.216,A -85,B 0,C 180,E1 5788.896,E2 5788.896} C_VEL
LIN {X 0,Y 182.121,Z 713.67,A -85,B 0,C 180,E1 5785.796,E2 5785.796} C_VEL
LIN {X 0,Y 193.227,Z 699.046,A -85,B 0,C 180,E1 5783.3,E2 5783.3} C_VEL
LIN {X 0,Y 203.313,Z 683.449,A -85,B 0,C 180,E1 5781.267,E2 5781.267} C_VEL
LIN {X 0,Y 212.707,Z 666.077,A -85,B 0,C 180,E1 5779.533,E2 5779.533} C_VEL
LIN {X 0,Y 220.463,Z 648.509,A -85,B 0,C 180,E1 5778.174,E2 5778.174} C_VEL
LIN {X 0,Y 226.951,Z 629.916,A -85,B 0,C 180,E1 5777.062,E2 5777.062} C_VEL
LIN {X 0,Y 231.994,Z 610.496,A -85,B 0,C 180,E1 5776.179,E2 5776.179} C_VEL
LIN {X 0,Y 235.428,Z 590.695,A -85,B 0,C 180,E1 5775.516,E2 5775.516} C_VEL
LIN {X 0,Y 240.775,Z 541.624,A -85,B 0,C 180,E1 5774.485,E2 5774.485} C_VEL
LIN {X 0,Y 244.244,Z 509.703,A -85,B 0,C 180,E1 5773.894,E2 5773.894} C_VEL
LIN {X 0,Y 242.548,Z 505.607,A -85,B 0,C 180,E1 5770.691,E2 5770.691} C_VEL
LIN {X 0,Y 241.356,Z 502.858,A -85,B 0,C 180,E1 5767.14,E2 5767.14} C_VEL
LIN {X 0,Y 240.832,Z 502.679,A -85,B 0,C 180,E1 5762.38,E2 5762.38} C_VEL
LIN {X 0,Y 240.997,Z 503.351,A -85,B 0,C 180,E1 5760.476,E2 5760.476} C_VEL
LIN {X 0,Y 241.725,Z 506.331,A -85,B 0,C 180,E1 5757.037,E2 5757.037} C_VEL
LIN {X 0,Y 242.963,Z 510.535,A -85,B 0,C 180,E1 5753.918,E2 5753.918} C_VEL
LIN {X 0,Y 243.972,Z 514.154,A -85,B 0,C 180,E1 5751.989,E2 5751.989} C_VEL
LIN {X 0,Y 233.511,Z 605.792,A -85,B 0,C 180,E1 5750.264,E2 5750.264} C_VEL
LIN {X 0,Y 229.253,Z 626.792,A -85,B 0,C 180,E1 5749.738,E2 5749.738} C_VEL
LIN {X 0,Y 223.491,Z 646.514,A -85,B 0,C 180,E1 5749.105,E2 5749.105} C_VEL
LIN {X 0,Y 215.959,Z 666.059,A -85,B 0,C 180,E1 5748.29,E2 5748.29} C_VEL
LIN {X 0,Y 206.616,Z 685.431,A -85,B 0,C 180,E1 5747.18,E2 5747.18} C_VEL
LIN {X 0,Y 196.033,Z 703.611,A -85,B 0,C 180,E1 5745.71,E2 5745.71} C_VEL
LIN {X 0,Y 184.308,Z 720.702,A -85,B 0,C 180,E1 5743.777,E2 5743.777} C_VEL
LIN {X 0,Y 171.587,Z 736.704,A -85,B 0,C 180,E1 5741.241,E2 5741.241} C_VEL
LIN {X 0,Y 158.492,Z 751.13,A -85,B 0,C 180,E1 5738.023,E2 5738.023} C_VEL
LIN {X 0,Y 151.738,Z 757.922,A -85,B 0,C 180,E1 5736.048,E2 5736.048} C_VEL
LIN {X 0,Y 146.355,Z 762.485,A -85,B 0,C 180,E1 5734.795,E2 5734.795} C_VEL
LIN {X 0,Y 130.468,Z 773.041,A -85,B 0,C 180,E1 5732.132,E2 5732.132} C_VEL
LIN {X 0,Y 125.033,Z 776.84,A -85,B 0,C 180,E1 5730.328,E2 5730.328} C_VEL
LIN {X 0,Y 113.061,Z 786.062,A -85,B 0,C 180,E1 5723.584,E2 5723.584} C_VEL
LIN {X 0,Y 102.404,Z 794.079,A -85,B 0,C 180,E1 5714.666,E2 5714.666} C_VEL
LIN {X 0,Y 94.429,Z 800.558,A -85,B 0,C 180,E1 5703.407,E2 5703.407} C_VEL
LIN {X 0,Y 90.457,Z 805.134,A -85,B 0,C 180,E1 5690.714,E2 5690.714} C_VEL
LIN {X 0,Y 90.51,Z 807.709,A -85,B 0,C 180,E1 5678.256,E2 5678.256} C_VEL
LIN {X 0,Y 92.096,Z 808.487,A -85,B 0,C 180,E1 5670,E2 5670} C_VEL
LIN {X 0,Y 90.353,Z 807.482,A -85,B 0,C 180,E1 5660.445,E2 5660.445} C_VEL
LIN {X 0,Y 90.668,Z 804.69,A -85,B 0,C 180,E1 5647.98,E2 5647.98} C_VEL
LIN {X 0,Y 94.735,Z 800.228,A -85,B 0,C 180,E1 5635.988,E2 5635.988} C_VEL
LIN {X 0,Y 102.896,Z 793.646,A -85,B 0,C 180,E1 5624.819,E2 5624.819} C_VEL
LIN {X 0,Y 114.323,Z 785.031,A -85,B 0,C 180,E1 5615.575,E2 5615.575} C_VEL
LIN {X 0,Y 127.475,Z 774.798,A -85,B 0,C 180,E1 5608.543,E2 5608.543} C_VEL
LIN {X 0,Y 141.412,Z 762.986,A -85,B 0,C 180,E1 5603.198,E2 5603.198} C_VEL
LIN {X 0,Y 155.665,Z 749.525,A -85,B 0,C 180,E1 5599.121,E2 5599.121} C_VEL
LIN {X 0,Y 168.843,Z 735.44,A -85,B 0,C 180,E1 5596.16,E2 5596.16} C_VEL
LIN {X 0,Y 181.722,Z 719.65,A -85,B 0,C 180,E1 5593.809,E2 5593.809} C_VEL
LIN {X 0,Y 193.747,Z 702.505,A -85,B 0,C 180,E1 5592,E2 5592} C_VEL
LIN {X 0,Y 204.486,Z 684.384,A -85,B 0,C 180,E1 5590.646,E2 5590.646} C_VEL
LIN {X 0,Y 213.978,Z 664.99,A -85,B 0,C 180,E1 5589.628,E2 5589.628} C_VEL
LIN {X 0,Y 221.617,Z 645.415,A -85,B 0,C 180,E1 5588.877,E2 5588.877} C_VEL
LIN {X 0,Y 227.701,Z 624.684,A -85,B 0,C 180,E1 5588.264,E2 5588.264} C_VEL
LIN {X 0,Y 231.906,Z 603.656,A -85,B 0,C 180,E1 5587.776,E2 5587.776} C_VEL
LIN {X 0,Y 241.705,Z 519.132,A -85,B 0,C 180,E1 5586.239,E2 5586.239} C_VEL
LIN {X 0,Y 240.66,Z 515.225,A -85,B 0,C 180,E1 5583.692,E2 5583.692} C_VEL
LIN {X 0,Y 240.023,Z 512.685,A -85,B 0,C 180,E1 5581.432,E2 5581.432} C_VEL
LIN {X 0,Y 239.616,Z 510.589,A -85,B 0,C 180,E1 5578.565,E2 5578.565} C_VEL
LIN {X 0,Y 239.776,Z 510.326,A -85,B 0,C 180,E1 5574.256,E2 5574.256} C_VEL
LIN {X 0,Y 240.297,Z 511.038,A -85,B 0,C 180,E1 5572.002,E2 5572.002} C_VEL
LIN {X 0,Y 241.622,Z 514.446,A -85,B 0,C 180,E1 5568.422,E2 5568.422} C_VEL
LIN {X 0,Y 241.932,Z 515.521,A -85,B 0,C 180,E1 5567.738,E2 5567.738} C_VEL
LIN {X 0,Y 234.064,Z 586.669,A -85,B 0,C 180,E1 5566.407,E2 5566.407} C_VEL
LIN {X 0,Y 231.001,Z 606.336,A -85,B 0,C 180,E1 5565.82,E2 5565.82} C_VEL
LIN {X 0,Y 226.379,Z 625.497,A -85,B 0,C 180,E1 5565.047,E2 5565.047} C_VEL
LIN {X 0,Y 220.41,Z 643.634,A -85,B 0,C 180,E1 5564.087,E2 5564.087} C_VEL
LIN {X 0,Y 212.472,Z 662.413,A -85,B 0,C 180,E1 5562.796,E2 5562.796} C_VEL
LIN {X 0,Y 203.269,Z 679.933,A -85,B 0,C 180,E1 5561.238,E2 5561.238} C_VEL
LIN {X 0,Y 192.929,Z 696.248,A -85,B 0,C 180,E1 5559.338,E2 5559.338} C_VEL
LIN {X 0,Y 181.209,Z 711.831,A -85,B 0,C 180,E1 5556.935,E2 5556.935} C_VEL
LIN {X 0,Y 168.67,Z 726.01,A -85,B 0,C 180,E1 5553.981,E2 5553.981} C_VEL
LIN {X 0,Y 155.439,Z 738.839,A -85,B 0,C 180,E1 5550.269,E2 5550.269} C_VEL
LIN {X 0,Y 142.568,Z 749.651,A -85,B 0,C 180,E1 5545.846,E2 5545.846} C_VEL
LIN {X 0,Y 129.813,Z 759.013,A -85,B 0,C 180,E1 5540.26,E2 5540.26} C_VEL
LIN {X 0,Y 117.984,Z 766.672,A -85,B 0,C 180,E1 5533.347,E2 5533.347} C_VEL
LIN {X 0,Y 107.423,Z 772.79,A -85,B 0,C 180,E1 5524.594,E2 5524.594} C_VEL
LIN {X 0,Y 99.483,Z 777.018,A -85,B 0,C 180,E1 5514.334,E2 5514.334} C_VEL
LIN {X 0,Y 94.558,Z 779.51,A -85,B 0,C 180,E1 5502.829,E2 5502.829} C_VEL
LIN {X 0,Y 92.84,Z 780.375,A -85,B 0,C 180,E1 5490.617,E2 5490.617} C_VEL
LIN {X 0,Y 94.075,Z 779.741,A -85,B 0,C 180,E1 5478.971,E2 5478.971} C_VEL
LIN {X 0,Y 98.502,Z 777.524,A -85,B 0,C 180,E1 5467.312,E2 5467.312} C_VEL
LIN {X 0,Y 105.995,Z 773.595,A -85,B 0,C 180,E1 5456.832,E2 5456.832} C_VEL
LIN {X 0,Y 115.617,Z 768.141,A -85,B 0,C 180,E1 5448.251,E2 5448.251} C_VEL
LIN {X 0,Y 127.201,Z 760.858,A -85,B 0,C 180,E1 5441.011,E2 5441.011} C_VEL
LIN {X 0,Y 139.58,Z 752.061,A -85,B 0,C 180,E1 5435.255,E2 5435.255} C_VEL
LIN {X 0,Y 152.261,Z 741.791,A -85,B 0,C 180,E1 5430.659,E2 5430.659} C_VEL
LIN {X 0,Y 164.867,Z 730.079,A -85,B 0,C 180,E1 5426.941,E2 5426.941} C_VEL
LIN {X 0,Y 177.156,Z 716.89,A -85,B 0,C 180,E1 5423.894,E2 5423.894} C_VEL
LIN {X 0,Y 188.428,Z 702.85,A -85,B 0,C 180,E1 5421.478,E2 5421.478} C_VEL
LIN {X 0,Y 198.855,Z 687.656,A -85,B 0,C 180,E1 5419.484,E2 5419.484} C_VEL
LIN {X 0,Y 208.453,Z 671.011,A -85,B 0,C 180,E1 5417.808,E2 5417.808} C_VEL
LIN {X 0,Y 216.817,Z 653.35,A -85,B 0,C 180,E1 5416.429,E2 5416.429} C_VEL
LIN {X 0,Y 223.891,Z 634.523,A -85,B 0,C 180,E1 5415.293,E2 5415.293} C_VEL
LIN {X 0,Y 229.505,Z 614.573,A -85,B 0,C 180,E1 5414.379,E2 5414.379} C_VEL
LIN {X 0,Y 233.386,Z 594.183,A -85,B 0,C 180,E1 5413.688,E2 5413.688} C_VEL
LIN {X 0,Y 238.385,Z 550.093,A -85,B 0,C 180,E1 5412.75,E2 5412.75} C_VEL
LIN {X 0,Y 242.226,Z 515.518,A -85,B 0,C 180,E1 5412.153,E2 5412.153} C_VEL
LIN {X 0,Y 241.163,Z 512.939,A -85,B 0,C 180,E1 5409.787,E2 5409.787} C_VEL
LIN {X 0,Y 240.324,Z 510.761,A -85,B 0,C 180,E1 5406.93,E2 5406.93} C_VEL
LIN {X 0,Y 239.857,Z 510.626,A -85,B 0,C 180,E1 5402.39,E2 5402.39} C_VEL
LIN {X 0,Y 239.975,Z 511.274,A -85,B 0,C 180,E1 5400.667,E2 5400.667} C_VEL
LIN {X 0,Y 240.597,Z 514.157,A -85,B 0,C 180,E1 5397.38,E2 5397.38} C_VEL
LIN {X 0,Y 241.615,Z 517.981,A -85,B 0,C 180,E1 5394.539,E2 5394.539} C_VEL
LIN {X 0,Y 241.929,Z 519.643,A -85,B 0,C 180,E1 5393.751,E2 5393.751} C_VEL
LIN {X 0,Y 231.976,Z 604.943,A -85,B 0,C 180,E1 5392.211,E2 5392.211} C_VEL
LIN {X 0,Y 227.648,Z 625.941,A -85,B 0,C 180,E1 5391.718,E2 5391.718} C_VEL
LIN {X 0,Y 221.622,Z 646.151,A -85,B 0,C 180,E1 5391.115,E2 5391.115} C_VEL
LIN {X 0,Y 213.982,Z 665.58,A -85,B 0,C 180,E1 5390.365,E2 5390.365} C_VEL
LIN {X 0,Y 204.49,Z 684.835,A -85,B 0,C 180,E1 5389.346,E2 5389.346} C_VEL
LIN {X 0,Y 193.865,Z 702.702,A -85,B 0,C 180,E1 5388.007,E2 5388.007} C_VEL
LIN {X 0,Y 182.183,Z 719.358,A -85,B 0,C 180,E1 5386.259,E2 5386.259} C_VEL
LIN {X 0,Y 168.917,Z 735.615,A -85,B 0,C 180,E1 5383.848,E2 5383.848} C_VEL
LIN {X 0,Y 155.583,Z 749.831,A -85,B 0,C 180,E1 5380.851,E2 5380.851} C_VEL
LIN {X 0,Y 141.417,Z 763.16,A -85,B 0,C 180,E1 5376.796,E2 5376.796} C_VEL
LIN {X 0,Y 127.309,Z 775.078,A -85,B 0,C 180,E1 5371.376,E2 5371.376} C_VEL
LIN {X 0,Y 125.033,Z 776.84,A -85,B 0,C 180,E1 5370.328,E2 5370.328} C_VEL
LIN {X 0,Y 119.644,Z 780.505,A -85,B 0,C 180,E1 5368.303,E2 5368.303} C_VEL
LIN {X 0,Y 103.917,Z 788.435,A -85,B 0,C 180,E1 5363.293,E2 5363.293} C_VEL
LIN {X 0,Y 98.999,Z 791.173,A -85,B 0,C 180,E1 5360.308,E2 5360.308} C_VEL
LIN {X 0,Y 89.495,Z 797.808,A -85,B 0,C 180,E1 5349.554,E2 5349.554} C_VEL
LIN {X 0,Y 83.509,Z 802.905,A -85,B 0,C 180,E1 5336.109,E2 5336.109} C_VEL
LIN {X 0,Y 82.208,Z 806.044,A -85,B 0,C 180,E1 5321.932,E2 5321.932} C_VEL
LIN {X 0,Y 83.991,Z 807.245,A -85,B 0,C 180,E1 5310.588,E2 5310.588} C_VEL
LIN {X 0,Y 83.384,Z 807.03,A -85,B 0,C 180,E1 5306.563,E2 5306.563} C_VEL
LIN {X 0,Y 82.141,Z 805.282,A -85,B 0,C 180,E1 5293.742,E2 5293.742} C_VEL
LIN {X 0,Y 84.867,Z 801.532,A -85,B 0,C 180,E1 5279.563,E2 5279.563} C_VEL
LIN {X 0,Y 92.102,Z 795.911,A -85,B 0,C 180,E1 5266.85,E2 5266.85} C_VEL
LIN {X 0,Y 103.09,Z 788.327,A -85,B 0,C 180,E1 5256.391,E2 5256.391} C_VEL
LIN {X 0,Y 116.107,Z 779.176,A -85,B 0,C 180,E1 5248.556,E2 5248.556} C_VEL
LIN {X 0,Y 130.823,Z 767.94,A -85,B 0,C 180,E1 5242.465,E2 5242.465} C_VEL
LIN {X 0,Y 145.187,Z 755.703,A -85,B 0,C 180,E1 5238.133,E2 5238.133} C_VEL
LIN {X 0,Y 159.305,Z 742.07,A -85,B 0,C 180,E1 5234.865,E2 5234.865} C_VEL
LIN {X 0,Y 173.069,Z 726.822,A -85,B 0,C 180,E1 5232.342,E2 5232.342} C_VEL
LIN {X 0,Y 186.032,Z 710.124,A -85,B 0,C 180,E1 5230.411,E2 5230.411} C_VEL
LIN {X 0,Y 197.404,Z 692.878,A -85,B 0,C 180,E1 5229.012,E2 5229.012} C_VEL
LIN {X 0,Y 207.467,Z 674.649,A -85,B 0,C 180,E1 5227.965,E2 5227.965} C_VEL
LIN {X 0,Y 216.181,Z 655.296,A -85,B 0,C 180,E1 5227.173,E2 5227.173} C_VEL
LIN {X 0,Y 223.171,Z 635.374,A -85,B 0,C 180,E1 5226.555,E2 5226.555} C_VEL
LIN {X 0,Y 228.427,Z 614.833,A -85,B 0,C 180,E1 5226.053,E2 5226.053} C_VEL
LIN {X 0,Y 231.864,Z 593.892,A -85,B 0,C 180,E1 5225.639,E2 5225.639} C_VEL
LIN {X 0,Y 239.884,Z 524.505,A -85,B 0,C 180,E1 5224.422,E2 5224.422} C_VEL
LIN {X 0,Y 238.911,Z 520.38,A -85,B 0,C 180,E1 5220.959,E2 5220.959} C_VEL
LIN {X 0,Y 238.604,Z 518.485,A -85,B 0,C 180,E1 5218.319,E2 5218.319} C_VEL
LIN {X 0,Y 238.836,Z 518.302,A -85,B 0,C 180,E1 5213.992,E2 5213.992} C_VEL
LIN {X 0,Y 239.254,Z 518.975,A -85,B 0,C 180,E1 5212.193,E2 5212.193} C_VEL
LIN {X 0,Y 240.118,Z 521.439,A -85,B 0,C 180,E1 5209.523,E2 5209.523} C_VEL
LIN {X 0,Y 232.606,Z 587.716,A -85,B 0,C 180,E1 5208.324,E2 5208.324} C_VEL
LIN {X 0,Y 229.46,Z 607.309,A -85,B 0,C 180,E1 5207.759,E2 5207.759} C_VEL
LIN {X 0,Y 224.707,Z 626.53,A -85,B 0,C 180,E1 5207.017,E2 5207.017} C_VEL
LIN {X 0,Y 218.386,Z 645.241,A -85,B 0,C 180,E1 5206.071,E2 5206.071} C_VEL
LIN {X 0,Y 210.187,Z 664.05,A -85,B 0,C 180,E1 5204.832,E2 5204.832} C_VEL
LIN {X 0,Y 200.873,Z 681.311,A -85,B 0,C 180,E1 5203.367,E2 5203.367} C_VEL
LIN {X 0,Y 190.245,Z 697.637,A -85,B 0,C 180,E1 5201.553,E2 5201.553} C_VEL
LIN {X 0,Y 178.045,Z 713.365,A -85,B 0,C 180,E1 5199.228,E2 5199.228} C_VEL
LIN {X 0,Y 165.69,Z 726.92,A -85,B 0,C 180,E1 5196.523,E2 5196.523} C_VEL
LIN {X 0,Y 152.473,Z 739.373,A -85,B 0,C 180,E1 5193.097,E2 5193.097} C_VEL
LIN {X 0,Y 138.83,Z 750.45,A -85,B 0,C 180,E1 5188.764,E2 5188.764} C_VEL
LIN {X 0,Y 125.006,Z 760.153,A -85,B 0,C 180,E1 5183.113,E2 5183.113} C_VEL
LIN {X 0,Y 112.346,Z 767.883,A -85,B 0,C 180,E1 5176.126,E2 5176.126} C_VEL
LIN {X 0,Y 100.993,Z 773.997,A -85,B 0,C 180,E1 5167.15,E2 5167.15} C_VEL
LIN {X 0,Y 92.317,Z 778.223,A -85,B 0,C 180,E1 5156.362,E2 5156.362} C_VEL
LIN {X 0,Y 86.856,Z 780.714,A -85,B 0,C 180,E1 5143.989,E2 5143.989} C_VEL
LIN {X 0,Y 84.931,Z 781.576,A -85,B 0,C 180,E1 5130.675,E2 5130.675} C_VEL
LIN {X 0,Y 86.318,Z 780.943,A -85,B 0,C 180,E1 5117.966,E2 5117.966} C_VEL
LIN {X 0,Y 91.239,Z 778.726,A -85,B 0,C 180,E1 5105.392,E2 5105.392} C_VEL
LIN {X 0,Y 99.448,Z 774.799,A -85,B 0,C 180,E1 5094.33,E2 5094.33} C_VEL
LIN {X 0,Y 109.825,Z 769.346,A -85,B 0,C 180,E1 5085.493,E2 5085.493} C_VEL
LIN {X 0,Y 122.142,Z 762.067,A -85,B 0,C 180,E1 5078.202,E2 5078.202} C_VEL
LIN {X 0,Y 135.159,Z 753.275,A -85,B 0,C 180,E1 5072.509,E2 5072.509} C_VEL
LIN {X 0,Y 149.179,Z 742.345,A -85,B 0,C 180,E1 5067.787,E2 5067.787} C_VEL
LIN {X 0,Y 162.268,Z 730.507,A -85,B 0,C 180,E1 5064.229,E2 5064.229} C_VEL
LIN {X 0,Y 174.96,Z 717.175,A -85,B 0,C 180,E1 5061.333,E2 5061.333} C_VEL
LIN {X 0,Y 186.668,Z 702.82,A -85,B 0,C 180,E1 5059.026,E2 5059.026} C_VEL
LIN {X 0,Y 197.251,Z 687.577,A -85,B 0,C 180,E1 5057.163,E2 5057.163} C_VEL
LIN {X 0,Y 206.628,Z 671.559,A -85,B 0,C 180,E1 5055.652,E2 5055.652} C_VEL
LIN {X 0,Y 215.174,Z 653.799,A -85,B 0,C 180,E1 5054.346,E2 5054.346} C_VEL
LIN {X 0,Y 222.239,Z 635.333,A -85,B 0,C 180,E1 5053.293,E2 5053.293} C_VEL
LIN {X 0,Y 227.976,Z 615.339,A -85,B 0,C 180,E1 5052.421,E2 5052.421} C_VEL
LIN {X 0,Y 231.933,Z 595.031,A -85,B 0,C 180,E1 5051.761,E2 5051.761} C_VEL
LIN {X 0,Y 237.074,Z 550.869,A -85,B 0,C 180,E1 5050.855,E2 5050.855} C_VEL
LIN {X 0,Y 240.401,Z 521.512,A -85,B 0,C 180,E1 5050.363,E2 5050.363} C_VEL
LIN {X 0,Y 239.297,Z 518.666,A -85,B 0,C 180,E1 5046.719,E2 5046.719} C_VEL
LIN {X 0,Y 238.877,Z 518.617,A -85,B 0,C 180,E1 5042.159,E2 5042.159} C_VEL
LIN {X 0,Y 238.985,Z 519.502,A -85,B 0,C 180,E1 5040.48,E2 5040.48} C_VEL
LIN {X 0,Y 239.478,Z 521.981,A -85,B 0,C 180,E1 5037.727,E2 5037.727} C_VEL
LIN {X 0,Y 240.149,Z 524.875,A -85,B 0,C 180,E1 5035.546,E2 5035.546} C_VEL
LIN {X 0,Y 230.682,Z 604.257,A -85,B 0,C 180,E1 5034.178,E2 5034.178} C_VEL
LIN {X 0,Y 226.318,Z 625.089,A -85,B 0,C 180,E1 5033.723,E2 5033.723} C_VEL
LIN {X 0,Y 220.273,Z 645.123,A -85,B 0,C 180,E1 5033.176,E2 5033.176} C_VEL
LIN {X 0,Y 212.775,Z 664.027,A -85,B 0,C 180,E1 5032.519,E2 5032.519} C_VEL
LIN {X 0,Y 203.143,Z 683.398,A -85,B 0,C 180,E1 5031.603,E2 5031.603} C_VEL
LIN {X 0,Y 192.175,Z 701.559,A -85,B 0,C 180,E1 5030.371,E2 5030.371} C_VEL
LIN {X 0,Y 179.943,Z 718.616,A -85,B 0,C 180,E1 5028.725,E2 5028.725} C_VEL
LIN {X 0,Y 166.558,Z 734.579,A -85,B 0,C 180,E1 5026.523,E2 5026.523} C_VEL
LIN {X 0,Y 152.184,Z 749.379,A -85,B 0,C 180,E1 5023.576,E2 5023.576} C_VEL
LIN {X 0,Y 137.513,Z 762.58,A -85,B 0,C 180,E1 5019.707,E2 5019.707} C_VEL
LIN {X 0,Y 122.935,Z 774.245,A -85,B 0,C 180,E1 5014.523,E2 5014.523} C_VEL
LIN {X 0,Y 108.994,Z 784.336,A -85,B 0,C 180,E1 5007.558,E2 5007.558} C_VEL
LIN {X 0,Y 98.999,Z 791.173,A -85,B 0,C 180,E1 5000.308,E2 5000.308} C_VEL
LIN {X 0,Y 94.331,Z 793.782,A -85,B 0,C 180,E1 4996.965,E2 4996.965} C_VEL
